LIN {X 0,Y 219.292,Z 411.491,A -85,B 0,C 180,E1 -21728.678,E2 -21728.678} C_VEL
LIN {X 0,Y 224.312,Z 397.889,A -85,B 0,C 180,E1 -21730.847,E2 -21730.847} C_VEL
LIN {X 0,Y 228.493,Z 384.244,A -85,B 0,C 180,E1 -21732.585,E2 -21732.585} C_VEL
LIN {X 0,Y 232.119,Z 370.098,A -85,B 0,C 180,E1 -21733.987,E2 -21733.987} C_VEL
LIN {X 0,Y 235.267,Z 355.521,A -85,B 0,C 180,E1 -21735.04,E2 -21735.04} C_VEL
LIN {X 0,Y 237.617,Z 340.528,A -85,B 0,C 180,E1 -21735.827,E2 -21735.827} C_VEL
LIN {X 0,Y 239.137,Z 325.025,A -85,B 0,C 180,E1 -21736.361,E2 -21736.361} C_VEL
LIN {X 0,Y 243.824,Z 251.846,A -85,B 0,C 180,E1 -21738.299,E2 -21738.299} C_VEL
LIN {X 0,Y 243.721,Z 250.513,A -85,B 0,C 180,E1 -21738.384,E2 -21738.384} C_VEL
LIN {X 0,Y 238.615,Z 238.715,A -85,B 0,C 180,E1 -21740.32,E2 -21740.32} C_VEL
LIN {X 0,Y 233.027,Z 227.32,A -85,B 0,C 180,E1 -21742.562,E2 -21742.562} C_VEL
LIN {X 0,Y 226.426,Z 215.296,A -85,B 0,C 180,E1 -21745.446,E2 -21745.446} C_VEL
LIN {X 0,Y 223.259,Z 210.38,A -85,B 0,C 180,E1 -21746.923,E2 -21746.923} C_VEL
LIN {X 0,Y 218.11,Z 203.18,A -85,B 0,C 180,E1 -21749.507,E2 -21749.507} C_VEL
LIN {X 0,Y 214.873,Z 198.917,A -85,B 0,C 180,E1 -21751.289,E2 -21751.289} C_VEL
LIN {X 0,Y 211.946,Z 195.104,A -85,B 0,C 180,E1 -21753.04,E2 -21753.04} C_VEL
LIN {X 0,Y 208.457,Z 191.041,A -85,B 0,C 180,E1 -21755.308,E2 -21755.308} C_VEL
LIN {X 0,Y 207.502,Z 189.433,A -85,B 0,C 180,E1 -21756.019,E2 -21756.019} C_VEL
LIN {X 0,Y 204.843,Z 187.038,A -85,B 0,C 180,E1 -21757.96,E2 -21757.96} C_VEL
LIN {X 0,Y 202.817,Z 183.879,A -85,B 0,C 180,E1 -21759.726,E2 -21759.726} C_VEL
LIN {X 0,Y 200.124,Z 181.801,A -85,B 0,C 180,E1 -21762.152,E2 -21762.152} C_VEL
LIN {X 0,Y 198.455,Z 178.926,A -85,B 0,C 180,E1 -21764.071,E2 -21764.071} C_VEL
LIN {X 0,Y 197.838,Z 178.138,A -85,B 0,C 180,E1 -21764.812,E2 -21764.812} C_VEL
LIN {X 0,Y 194.773,Z 176.058,A -85,B 0,C 180,E1 -21768.949,E2 -21768.949} C_VEL
LIN {X 0,Y 193.148,Z 172.89,A -85,B 0,C 180,E1 -21772.946,E2 -21772.946} C_VEL
LIN {X 0,Y 193.084,Z 172.118,A -85,B 0,C 180,E1 -21776.87,E2 -21776.87} C_VEL
LIN {X 0,Y 193.435,Z 172.028,A -85,B 0,C 180,E1 -21780,E2 -21780} C_VEL
LIN {X 0,Y 192.969,Z 172.206,A -85,B 0,C 180,E1 -21784.177,E2 -21784.177} C_VEL
LIN {X 0,Y 193.221,Z 173.073,A -85,B 0,C 180,E1 -21787.577,E2 -21787.577} C_VEL
LIN {X 0,Y 195.21,Z 176.548,A -85,B 0,C 180,E1 -21791.948,E2 -21791.948} C_VEL
LIN {X 0,Y 198.274,Z 178.589,A -85,B 0,C 180,E1 -21795.879,E2 -21795.879} C_VEL
LIN {X 0,Y 200,Z 181.766,A -85,B 0,C 180,E1 -21797.911,E2 -21797.911} C_VEL
LIN {X 0,Y 203.141,Z 184.315,A -85,B 0,C 180,E1 -21800.738,E2 -21800.738} C_VEL
LIN {X 0,Y 205.283,Z 187.689,A -85,B 0,C 180,E1 -21802.575,E2 -21802.575} C_VEL
LIN {X 0,Y 207.751,Z 189.895,A -85,B 0,C 180,E1 -21804.349,E2 -21804.349} C_VEL
LIN {X 0,Y 210.168,Z 193.303,A -85,B 0,C 180,E1 -21806.034,E2 -21806.034} C_VEL
LIN {X 0,Y 211.927,Z 195.13,A -85,B 0,C 180,E1 -21807.128,E2 -21807.128} C_VEL
LIN {X 0,Y 214.824,Z 198.894,A -85,B 0,C 180,E1 -21808.862,E2 -21808.862} C_VEL
LIN {X 0,Y 219.389,Z 204.99,A -85,B 0,C 180,E1 -21811.343,E2 -21811.343} C_VEL
LIN {X 0,Y 225.014,Z 212.914,A -85,B 0,C 180,E1 -21814.074,E2 -21814.074} C_VEL
LIN {X 0,Y 231.75,Z 223.28,A -85,B 0,C 180,E1 -21816.998,E2 -21816.998} C_VEL
LIN {X 0,Y 236.546,Z 232.253,A -85,B 0,C 180,E1 -21818.945,E2 -21818.945} C_VEL
LIN {X 0,Y 242.757,Z 245.504,A -85,B 0,C 180,E1 -21821.317,E2 -21821.317} C_VEL
LIN {X 0,Y 243.976,Z 248.447,A -85,B 0,C 180,E1 -21821.77,E2 -21821.77} C_VEL
LIN {X 0,Y 238.681,Z 329.958,A -85,B 0,C 180,E1 -21823.981,E2 -21823.981} C_VEL
LIN {X 0,Y 236.71,Z 345.1,A -85,B 0,C 180,E1 -21824.632,E2 -21824.632} C_VEL
LIN {X 0,Y 233.757,Z 361,A -85,B 0,C 180,E1 -21825.651,E2 -21825.651} C_VEL
LIN {X 0,Y 230.664,Z 374.454,A -85,B 0,C 180,E1 -21826.841,E2 -21826.841} C_VEL
LIN {X 0,Y 226.549,Z 389.137,A -85,B 0,C 180,E1 -21828.535,E2 -21828.535} C_VEL
LIN {X 0,Y 222.072,Z 402.265,A -85,B 0,C 180,E1 -21830.439,E2 -21830.439} C_VEL
LIN {X 0,Y 217.336,Z 414.499,A -85,B 0,C 180,E1 -21832.676,E2 -21832.676} C_VEL
LIN {X 0,Y 212.546,Z 425.648,A -85,B 0,C 180,E1 -21835.223,E2 -21835.223} C_VEL
LIN {X 0,Y 208.325,Z 435.023,A -85,B 0,C 180,E1 -21837.904,E2 -21837.904} C_VEL
LIN {X 0,Y 204.44,Z 443.018,A -85,B 0,C 180,E1 -21840.668,E2 -21840.668} C_VEL
LIN {X 0,Y 200.016,Z 451.913,A -85,B 0,C 180,E1 -21844.505,E2 -21844.505} C_VEL
LIN {X 0,Y 196.286,Z 459.241,A -85,B 0,C 180,E1 -21848.581,E2 -21848.581} C_VEL
LIN {X 0,Y 194.063,Z 464.117,A -85,B 0,C 180,E1 -21852.072,E2 -21852.072} C_VEL
LIN {X 0,Y 192.41,Z 467.578,A -85,B 0,C 180,E1 -21855.186,E2 -21855.186} C_VEL
LIN {X 0,Y 191.035,Z 471.08,A -85,B 0,C 180,E1 -21859.4,E2 -21859.4} C_VEL
LIN {X 0,Y 190.302,Z 473.393,A -85,B 0,C 180,E1 -21863.639,E2 -21863.639} C_VEL
LIN {X 0,Y 190.123,Z 474.569,A -85,B 0,C 180,E1 -21867.882,E2 -21867.882} C_VEL
LIN {X 0,Y 190.157,Z 474.726,A -85,B 0,C 180,E1 -21870,E2 -21870} C_VEL
LIN {X 0,Y 190.164,Z 474.157,A -85,B 0,C 180,E1 -21874.239,E2 -21874.239} C_VEL
LIN {X 0,Y 190.571,Z 472.465,A -85,B 0,C 180,E1 -21878.483,E2 -21878.483} C_VEL
LIN {X 0,Y 191.615,Z 469.61,A -85,B 0,C 180,E1 -21882.713,E2 -21882.713} C_VEL
LIN {X 0,Y 193.44,Z 465.523,A -85,B 0,C 180,E1 -21886.897,E2 -21886.897} C_VEL
LIN {X 0,Y 196.018,Z 460.105,A -85,B 0,C 180,E1 -21891.011,E2 -21891.011} C_VEL
LIN {X 0,Y 199.457,Z 453.203,A -85,B 0,C 180,E1 -21895.013,E2 -21895.013} C_VEL
LIN {X 0,Y 203.743,Z 444.589,A -85,B 0,C 180,E1 -21898.877,E2 -21898.877} C_VEL
LIN {X 0,Y 207.557,Z 436.846,A -85,B 0,C 180,E1 -21901.658,E2 -21901.658} C_VEL
LIN {X 0,Y 211.732,Z 427.731,A -85,B 0,C 180,E1 -21904.352,E2 -21904.352} C_VEL
LIN {X 0,Y 216.41,Z 416.978,A -85,B 0,C 180,E1 -21906.927,E2 -21906.927} C_VEL
LIN {X 0,Y 221.049,Z 405.24,A -85,B 0,C 180,E1 -21909.191,E2 -21909.191} C_VEL
LIN {X 0,Y 225.472,Z 392.675,A -85,B 0,C 180,E1 -21911.13,E2 -21911.13} C_VEL
LIN {X 0,Y 229.623,Z 378.937,A -85,B 0,C 180,E1 -21912.808,E2 -21912.808} C_VEL
LIN {X 0,Y 233.12,Z 364.473,A -85,B 0,C 180,E1 -21914.2,E2 -21914.2} C_VEL
LIN {X 0,Y 236.194,Z 349.03,A -85,B 0,C 180,E1 -21915.268,E2 -21915.268} C_VEL
LIN {X 0,Y 238.405,Z 333.558,A -85,B 0,C 180,E1 -21916.012,E2 -21916.012} C_VEL
LIN {X 0,Y 239.996,Z 314.021,A -85,B 0,C 180,E1 -21916.603,E2 -21916.603} C_VEL
LIN {X 0,Y 244.143,Z 248.635,A -85,B 0,C 180,E1 -21918.345,E2 -21918.345} C_VEL
LIN {X 0,Y 238.871,Z 236.861,A -85,B 0,C 180,E1 -21920.33,E2 -21920.33} C_VEL
LIN {X 0,Y 232.951,Z 225.151,A -85,B 0,C 180,E1 -21922.702,E2 -21922.702} C_VEL
LIN {X 0,Y 226.627,Z 215.259,A -85,B 0,C 180,E1 -21925.396,E2 -21925.396} C_VEL
LIN {X 0,Y 220.963,Z 207.127,A -85,B 0,C 180,E1 -21928.077,E2 -21928.077} C_VEL
LIN {X 0,Y 217.799,Z 202.785,A -85,B 0,C 180,E1 -21929.718,E2 -21929.718} C_VEL
LIN {X 0,Y 214.768,Z 198.812,A -85,B 0,C 180,E1 -21931.407,E2 -21931.407} C_VEL
LIN {X 0,Y 211.862,Z 194.934,A -85,B 0,C 180,E1 -21933.171,E2 -21933.171} C_VEL
LIN {X 0,Y 208.527,Z 191.176,A -85,B 0,C 180,E1 -21935.35,E2 -21935.35} C_VEL
LIN {X 0,Y 207.444,Z 189.425,A -85,B 0,C 180,E1 -21936.158,E2 -21936.158} C_VEL
LIN {X 0,Y 204.828,Z 187.087,A -85,B 0,C 180,E1 -21938.09,E2 -21938.09} C_VEL
LIN {X 0,Y 202.979,Z 183.958,A -85,B 0,C 180,E1 -21939.742,E2 -21939.742} C_VEL
LIN {X 0,Y 200.155,Z 181.908,A -85,B 0,C 180,E1 -21942.302,E2 -21942.302} C_VEL
LIN {X 0,Y 198.377,Z 178.846,A -85,B 0,C 180,E1 -21944.393,E2 -21944.393} C_VEL
LIN {X 0,Y 197.616,Z 178.027,A -85,B 0,C 180,E1 -21945.321,E2 -21945.321} C_VEL
LIN {X 0,Y 194.83,Z 176.101,A -85,B 0,C 180,E1 -21949.255,E2 -21949.255} C_VEL
LIN {X 0,Y 193.129,Z 172.939,A -85,B 0,C 180,E1 -21953.732,E2 -21953.732} C_VEL
LIN {X 0,Y 193.236,Z 172.108,A -85,B 0,C 180,E1 -21957.915,E2 -21957.915} C_VEL
LIN {X 0,Y 193.433,Z 172.045,A -85,B 0,C 180,E1 -21960,E2 -21960} C_VEL
LIN {X 0,Y 193.021,Z 172.37,A -85,B 0,C 180,E1 -21964.176,E2 -21964.176} C_VEL
LIN {X 0,Y 193.222,Z 173.274,A -85,B 0,C 180,E1 -21966.789,E2 -21966.789} C_VEL
LIN {X 0,Y 195.939,Z 177.12,A -85,B 0,C 180,E1 -21972.428,E2 -21972.428} C_VEL
LIN {X 0,Y 198.359,Z 178.653,A -85,B 0,C 180,E1 -21975.476,E2 -21975.476} C_VEL
LIN {X 0,Y 200.006,Z 181.652,A -85,B 0,C 180,E1 -21977.447,E2 -21977.447} C_VEL
LIN {X 0,Y 202.504,Z 183.704,A -85,B 0,C 180,E1 -21979.778,E2 -21979.778} C_VEL
LIN {X 0,Y 203.192,Z 184.29,A -85,B 0,C 180,E1 -21980.367,E2 -21980.367} C_VEL
LIN {X 0,Y 205.214,Z 187.529,A -85,B 0,C 180,E1 -21982.13,E2 -21982.13} C_VEL
LIN {X 0,Y 207.902,Z 189.993,A -85,B 0,C 180,E1 -21984.087,E2 -21984.087} C_VEL
LIN {X 0,Y 210.279,Z 193.339,A -85,B 0,C 180,E1 -21985.753,E2 -21985.753} C_VEL
LIN {X 0,Y 212.074,Z 195.266,A -85,B 0,C 180,E1 -21986.88,E2 -21986.88} C_VEL
LIN {X 0,Y 215.083,Z 199.099,A -85,B 0,C 180,E1 -21988.68,E2 -21988.68} C_VEL
LIN {X 0,Y 219.591,Z 205.175,A -85,B 0,C 180,E1 -21991.136,E2 -21991.136} C_VEL
LIN {X 0,Y 224.74,Z 212.412,A -85,B 0,C 180,E1 -21993.652,E2 -21993.652} C_VEL
LIN {X 0,Y 230.647,Z 222.756,A -85,B 0,C 180,E1 -21996.329,E2 -21996.329} C_VEL
LIN {X 0,Y 230.842,Z 223.057,A -85,B 0,C 180,E1 -21996.41,E2 -21996.41} C_VEL
LIN {X 0,Y 232.605,Z 227.635,A -85,B 0,C 180,E1 -21997.223,E2 -21997.223} C_VEL
LIN {X 0,Y 234.592,Z 236.333,A -85,B 0,C 180,E1 -21998.279,E2 -21998.279} C_VEL
LIN {X 0,Y 236.857,Z 247.053,A -85,B 0,C 180,E1 -21999.47,E2 -21999.47} C_VEL
LIN {X 0,Y 237.942,Z 250.365,A -85,B 0,C 180,E1 -21999.938,E2 -21999.938} C_VEL
LIN {X 0,Y 239.15,Z 253.343,A -85,B 0,C 180,E1 -22000.418,E2 -22000.418} C_VEL
LIN {X 0,Y 234.71,Z 321.37,A -85,B 0,C 180,E1 -22002.254,E2 -22002.254} C_VEL
LIN {X 0,Y 233.155,Z 338.204,A -85,B 0,C 180,E1 -22002.794,E2 -22002.794} C_VEL
LIN {X 0,Y 230.899,Z 353.15,A -85,B 0,C 180,E1 -22003.548,E2 -22003.548} C_VEL
LIN {X 0,Y 227.895,Z 367.197,A -85,B 0,C 180,E1 -22004.508,E2 -22004.508} C_VEL
LIN {X 0,Y 224.313,Z 381.084,A -85,B 0,C 180,E1 -22005.803,E2 -22005.803} C_VEL
LIN {X 0,Y 220.1,Z 394.817,A -85,B 0,C 180,E1 -22007.474,E2 -22007.474} C_VEL
LIN {X 0,Y 215.197,Z 408.195,A -85,B 0,C 180,E1 -22009.527,E2 -22009.527} C_VEL
LIN {X 0,Y 210.282,Z 419.992,A -85,B 0,C 180,E1 -22011.807,E2 -22011.807} C_VEL
LIN {X 0,Y 205.38,Z 430.801,A -85,B 0,C 180,E1 -22014.427,E2 -22014.427} C_VEL
LIN {X 0,Y 200.245,Z 441.405,A -85,B 0,C 180,E1 -22017.674,E2 -22017.674} C_VEL
LIN {X 0,Y 195.813,Z 450.086,A -85,B 0,C 180,E1 -22021.018,E2 -22021.018} C_VEL
LIN {X 0,Y 192.484,Z 456.43,A -85,B 0,C 180,E1 -22024.014,E2 -22024.014} C_VEL
LIN {X 0,Y 188.856,Z 463.389,A -85,B 0,C 180,E1 -22028.152,E2 -22028.152} C_VEL
LIN {X 0,Y 186.229,Z 468.861,A -85,B 0,C 180,E1 -22032.428,E2 -22032.428} C_VEL
LIN {X 0,Y 184.342,Z 472.997,A -85,B 0,C 180,E1 -22036.776,E2 -22036.776} C_VEL
LIN {X 0,Y 183.382,Z 475.897,A -85,B 0,C 180,E1 -22041.182,E2 -22041.182} C_VEL
LIN {X 0,Y 183.012,Z 477.625,A -85,B 0,C 180,E1 -22045.595,E2 -22045.595} C_VEL
LIN {X 0,Y 183.058,Z 478.215,A -85,B 0,C 180,E1 -22050,E2 -22050} C_VEL
LIN {X 0,Y 183.012,Z 477.609,A -85,B 0,C 180,E1 -22054.405,E2 -22054.405} C_VEL
LIN {X 0,Y 183.381,Z 475.859,A -85,B 0,C 180,E1 -22058.818,E2 -22058.818} C_VEL
LIN {X 0,Y 184.332,Z 472.943,A -85,B 0,C 180,E1 -22063.224,E2 -22063.224} C_VEL
LIN {X 0,Y 186.211,Z 468.793,A -85,B 0,C 180,E1 -22067.574,E2 -22067.574} C_VEL
LIN {X 0,Y 188.83,Z 463.295,A -85,B 0,C 180,E1 -22071.851,E2 -22071.851} C_VEL
LIN {X 0,Y 192.475,Z 456.304,A -85,B 0,C 180,E1 -22075.987,E2 -22075.987} C_VEL
LIN {X 0,Y 196.458,Z 448.827,A -85,B 0,C 180,E1 -22079.465,E2 -22079.465} C_VEL
LIN {X 0,Y 200.307,Z 440.84,A -85,B 0,C 180,E1 -22082.49,E2 -22082.49} C_VEL
LIN {X 0,Y 205.393,Z 430.604,A -85,B 0,C 180,E1 -22085.57,E2 -22085.57} C_VEL
LIN {X 0,Y 210.304,Z 419.758,A -85,B 0,C 180,E1 -22088.188,E2 -22088.188} C_VEL
LIN {X 0,Y 215.163,Z 407.916,A -85,B 0,C 180,E1 -22090.48,E2 -22090.48} C_VEL
LIN {X 0,Y 220.112,Z 394.443,A -85,B 0,C 180,E1 -22092.529,E2 -22092.529} C_VEL
LIN {X 0,Y 224.29,Z 380.638,A -85,B 0,C 180,E1 -22094.202,E2 -22094.202} C_VEL
LIN {X 0,Y 227.856,Z 366.64,A -85,B 0,C 180,E1 -22095.501,E2 -22095.501} C_VEL
LIN {X 0,Y 230.97,Z 351.645,A -85,B 0,C 180,E1 -22096.512,E2 -22096.512} C_VEL
LIN {X 0,Y 233.166,Z 337.075,A -85,B 0,C 180,E1 -22097.203,E2 -22097.203} C_VEL
LIN {X 0,Y 234.769,Z 317.786,A -85,B 0,C 180,E1 -22097.809,E2 -22097.809} C_VEL
LIN {X 0,Y 239.057,Z 253.811,A -85,B 0,C 180,E1 -22099.505,E2 -22099.505} C_VEL
LIN {X 0,Y 237.375,Z 249.287,A -85,B 0,C 180,E1 -22100.19,E2 -22100.19} C_VEL
LIN {X 0,Y 231.82,Z 236.957,A -85,B 0,C 180,E1 -22102.47,E2 -22102.47} C_VEL
LIN {X 0,Y 225.569,Z 224.712,A -85,B 0,C 180,E1 -22105.245,E2 -22105.245} C_VEL
LIN {X 0,Y 220.942,Z 216.873,A -85,B 0,C 180,E1 -22107.468,E2 -22107.468} C_VEL
LIN {X 0,Y 215.767,Z 209.397,A -85,B 0,C 180,E1 -22110.168,E2 -22110.168} C_VEL
LIN {X 0,Y 212.349,Z 204.879,A -85,B 0,C 180,E1 -22112.129,E2 -22112.129} C_VEL
LIN {X 0,Y 209.047,Z 200.53,A -85,B 0,C 180,E1 -22114.218,E2 -22114.218} C_VEL
LIN {X 0,Y 206.284,Z 197.099,A -85,B 0,C 180,E1 -22116.136,E2 -22116.136} C_VEL
LIN {X 0,Y 205.372,Z 195.826,A -85,B 0,C 180,E1 -22116.825,E2 -22116.825} C_VEL
LIN {X 0,Y 202.634,Z 192.917,A -85,B 0,C 180,E1 -22118.976,E2 -22118.976} C_VEL
LIN {X 0,Y 201.143,Z 190.555,A -85,B 0,C 180,E1 -22120.349,E2 -22120.349} C_VEL
LIN {X 0,Y 198.576,Z 188.38,A -85,B 0,C 180,E1 -22122.786,E2 -22122.786} C_VEL
LIN {X 0,Y 196.671,Z 185.074,A -85,B 0,C 180,E1 -22125.117,E2 -22125.117} C_VEL
LIN {X 0,Y 193.651,Z 182.936,A -85,B 0,C 180,E1 -22129.347,E2 -22129.347} C_VEL
LIN {X 0,Y 191.942,Z 179.766,A -85,B 0,C 180,E1 -22133.43,E2 -22133.43} C_VEL
LIN {X 0,Y 190.91,Z 178.77,A -85,B 0,C 180,E1 -22137.891,E2 -22137.891} C_VEL
LIN {X 0,Y 190.889,Z 178.767,A -85,B 0,C 180,E1 -22142.11,E2 -22142.11} C_VEL
LIN {X 0,Y 192.003,Z 179.832,A -85,B 0,C 180,E1 -22146.921,E2 -22146.921} C_VEL
LIN {X 0,Y 194.313,Z 183.638,A -85,B 0,C 180,E1 -22151.937,E2 -22151.937} C_VEL
LIN {X 0,Y 196.86,Z 185.396,A -85,B 0,C 180,E1 -22155.307,E2 -22155.307} C_VEL
LIN {X 0,Y 198.783,Z 188.745,A -85,B 0,C 180,E1 -22157.624,E2 -22157.624} C_VEL
LIN {X 0,Y 201.508,Z 191.037,A -85,B 0,C 180,E1 -22160.164,E2 -22160.164} C_VEL
LIN {X 0,Y 203.775,Z 194.502,A -85,B 0,C 180,E1 -22162.162,E2 -22162.162} C_VEL
LIN {X 0,Y 205.859,Z 196.44,A -85,B 0,C 180,E1 -22163.717,E2 -22163.717} C_VEL
LIN {X 0,Y 208.564,Z 200.115,A -85,B 0,C 180,E1 -22165.65,E2 -22165.65} C_VEL
LIN {X 0,Y 209.923,Z 201.694,A -85,B 0,C 180,E1 -22166.535,E2 -22166.535} C_VEL
LIN {X 0,Y 213.72,Z 206.734,A -85,B 0,C 180,E1 -22168.86,E2 -22168.86} C_VEL
LIN {X 0,Y 217.46,Z 211.932,A -85,B 0,C 180,E1 -22170.935,E2 -22170.935} C_VEL
LIN {X 0,Y 222.021,Z 218.436,A -85,B 0,C 180,E1 -22173.232,E2 -22173.232} C_VEL
LIN {X 0,Y 228.588,Z 228.837,A -85,B 0,C 180,E1 -22176.22,E2 -22176.22} C_VEL
LIN {X 0,Y 232.998,Z 237.37,A -85,B 0,C 180,E1 -22178.1,E2 -22178.1} C_VEL
LIN {X 0,Y 238.901,Z 250.316,A -85,B 0,C 180,E1 -22180.469,E2 -22180.469} C_VEL
LIN {X 0,Y 239.153,Z 251.863,A -85,B 0,C 180,E1 -22180.61,E2 -22180.61} C_VEL
LIN {X 0,Y 233.807,Z 330.039,A -85,B 0,C 180,E1 -22182.729,E2 -22182.729} C_VEL
LIN {X 0,Y 231.659,Z 345.951,A -85,B 0,C 180,E1 -22183.431,E2 -22183.431} C_VEL
LIN {X 0,Y 228.733,Z 361.074,A -85,B 0,C 180,E1 -22184.408,E2 -22184.408} C_VEL
LIN {X 0,Y 225.536,Z 374.526,A -85,B 0,C 180,E1 -22185.607,E2 -22185.607} C_VEL
LIN {X 0,Y 221.613,Z 388.162,A -85,B 0,C 180,E1 -22187.18,E2 -22187.18} C_VEL
LIN {X 0,Y 217.098,Z 401.091,A -85,B 0,C 180,E1 -22189.039,E2 -22189.039} C_VEL
LIN {X 0,Y 212.119,Z 413.53,A -85,B 0,C 180,E1 -22191.29,E2 -22191.29} C_VEL
LIN {X 0,Y 207.508,Z 423.947,A -85,B 0,C 180,E1 -22193.651,E2 -22193.651} C_VEL
LIN {X 0,Y 202.936,Z 433.612,A -85,B 0,C 180,E1 -22196.351,E2 -22196.351} C_VEL
LIN {X 0,Y 198.947,Z 441.859,A -85,B 0,C 180,E1 -22199.188,E2 -22199.188} C_VEL
LIN {X 0,Y 194.682,Z 449.971,A -85,B 0,C 180,E1 -22202.595,E2 -22202.595} C_VEL
LIN {X 0,Y 191.095,Z 456.666,A -85,B 0,C 180,E1 -22206.137,E2 -22206.137} C_VEL
LIN {X 0,Y 187.879,Z 462.862,A -85,B 0,C 180,E1 -22210.326,E2 -22210.326} C_VEL
LIN {X 0,Y 185.512,Z 467.646,A -85,B 0,C 180,E1 -22214.622,E2 -22214.622} C_VEL
LIN {X 0,Y 184.04,Z 471.147,A -85,B 0,C 180,E1 -22218.993,E2 -22218.993} C_VEL
LIN {X 0,Y 183.232,Z 473.46,A -85,B 0,C 180,E1 -22223.393,E2 -22223.393} C_VEL
LIN {X 0,Y 183.041,Z 474.636,A -85,B 0,C 180,E1 -22227.8,E2 -22227.8} C_VEL
LIN {X 0,Y 183.068,Z 474.792,A -85,B 0,C 180,E1 -22230,E2 -22230} C_VEL
LIN {X 0,Y 183.078,Z 474.223,A -85,B 0,C 180,E1 -22234.403,E2 -22234.403} C_VEL
LIN {X 0,Y 183.534,Z 472.531,A -85,B 0,C 180,E1 -22238.811,E2 -22238.811} C_VEL
LIN {X 0,Y 184.668,Z 469.676,A -85,B 0,C 180,E1 -22243.2,E2 -22243.2} C_VEL
LIN {X 0,Y 186.615,Z 465.588,A -85,B 0,C 180,E1 -22247.535,E2 -22247.535} C_VEL
LIN {X 0,Y 189.53,Z 459.81,A -85,B 0,C 180,E1 -22252.023,E2 -22252.023} C_VEL
LIN {X 0,Y 192.992,Z 453.268,A -85,B 0,C 180,E1 -22255.912,E2 -22255.912} C_VEL
LIN {X 0,Y 197.525,Z 444.654,A -85,B 0,C 180,E1 -22259.876,E2 -22259.876} C_VEL
LIN {X 0,Y 200.862,Z 438.293,A -85,B 0,C 180,E1 -22262.234,E2 -22262.234} C_VEL
LIN {X 0,Y 205.126,Z 429.42,A -85,B 0,C 180,E1 -22265.021,E2 -22265.021} C_VEL
LIN {X 0,Y 209.92,Z 418.99,A -85,B 0,C 180,E1 -22267.662,E2 -22267.662} C_VEL
LIN {X 0,Y 214.708,Z 407.645,A -85,B 0,C 180,E1 -22269.97,E2 -22269.97} C_VEL
LIN {X 0,Y 219.302,Z 395.318,A -85,B 0,C 180,E1 -22271.989,E2 -22271.989} C_VEL
LIN {X 0,Y 223.648,Z 381.836,A -85,B 0,C 180,E1 -22273.736,E2 -22273.736} C_VEL
LIN {X 0,Y 227.334,Z 367.862,A -85,B 0,C 180,E1 -22275.163,E2 -22275.163} C_VEL
LIN {X 0,Y 230.476,Z 353.504,A -85,B 0,C 180,E1 -22276.246,E2 -22276.246} C_VEL
LIN {X 0,Y 233.017,Z 338.009,A -85,B 0,C 180,E1 -22277.084,E2 -22277.084} C_VEL
LIN {X 0,Y 234.572,Z 322.858,A -85,B 0,C 180,E1 -22277.623,E2 -22277.623} C_VEL
LIN {X 0,Y 239.359,Z 251.323,A -85,B 0,C 180,E1 -22279.529,E2 -22279.529} C_VEL
LIN {X 0,Y 234.599,Z 240.563,A -85,B 0,C 180,E1 -22281.428,E2 -22281.428} C_VEL
LIN {X 0,Y 229.419,Z 230.11,A -85,B 0,C 180,E1 -22283.621,E2 -22283.621} C_VEL
LIN {X 0,Y 223.515,Z 220.68,A -85,B 0,C 180,E1 -22286.263,E2 -22286.263} C_VEL
LIN {X 0,Y 218.485,Z 213.239,A -85,B 0,C 180,E1 -22288.755,E2 -22288.755} C_VEL
LIN {X 0,Y 215.01,Z 208.427,A -85,B 0,C 180,E1 -22290.639,E2 -22290.639} C_VEL
LIN {X 0,Y 212.443,Z 204.96,A -85,B 0,C 180,E1 -22292.142,E2 -22292.142} C_VEL
LIN {X 0,Y 209.155,Z 200.66,A -85,B 0,C 180,E1 -22294.232,E2 -22294.232} C_VEL
LIN {X 0,Y 206.371,Z 197.247,A -85,B 0,C 180,E1 -22296.173,E2 -22296.173} C_VEL
LIN {X 0,Y 205.346,Z 195.837,A -85,B 0,C 180,E1 -22296.954,E2 -22296.954} C_VEL
LIN {X 0,Y 202.705,Z 193.053,A -85,B 0,C 180,E1 -22299.05,E2 -22299.05} C_VEL
LIN {X 0,Y 201.308,Z 190.663,A -85,B 0,C 180,E1 -22300.365,E2 -22300.365} C_VEL
LIN {X 0,Y 198.655,Z 188.536,A -85,B 0,C 180,E1 -22302.897,E2 -22302.897} C_VEL
LIN {X 0,Y 196.771,Z 185.147,A -85,B 0,C 180,E1 -22305.257,E2 -22305.257} C_VEL
LIN {X 0,Y 193.774,Z 183.052,A -85,B 0,C 180,E1 -22309.552,E2 -22309.552} C_VEL
LIN {X 0,Y 191.949,Z 179.786,A -85,B 0,C 180,E1 -22314.221,E2 -22314.221} C_VEL
LIN {X 0,Y 191.221,Z 178.897,A -85,B 0,C 180,E1 -22317.893,E2 -22317.893} C_VEL
LIN {X 0,Y 191.232,Z 178.897,A -85,B 0,C 180,E1 -22322.106,E2 -22322.106} C_VEL
LIN {X 0,Y 192.125,Z 180.108,A -85,B 0,C 180,E1 -22326.3,E2 -22326.3} C_VEL
LIN {X 0,Y 194.911,Z 184.113,A -85,B 0,C 180,E1 -22332.23,E2 -22332.23} C_VEL
LIN {X 0,Y 196.933,Z 185.341,A -85,B 0,C 180,E1 -22334.862,E2 -22334.862} C_VEL
LIN {X 0,Y 198.609,Z 188.405,A -85,B 0,C 180,E1 -22336.957,E2 -22336.957} C_VEL
LIN {X 0,Y 201.013,Z 190.483,A -85,B 0,C 180,E1 -22339.293,E2 -22339.293} C_VEL
LIN {X 0,Y 201.736,Z 191.396,A -85,B 0,C 180,E1 -22339.962,E2 -22339.962} C_VEL
LIN {X 0,Y 204.215,Z 194.854,A -85,B 0,C 180,E1 -22342.111,E2 -22342.111} C_VEL
LIN {X 0,Y 206.063,Z 196.647,A -85,B 0,C 180,E1 -22343.494,E2 -22343.494} C_VEL
LIN {X 0,Y 208.755,Z 200.236,A -85,B 0,C 180,E1 -22345.419,E2 -22345.419} C_VEL
LIN {X 0,Y 210.208,Z 201.994,A -85,B 0,C 180,E1 -22346.372,E2 -22346.372} C_VEL
LIN {X 0,Y 213.833,Z 206.786,A -85,B 0,C 180,E1 -22348.595,E2 -22348.595} C_VEL
LIN {X 0,Y 217.456,Z 211.781,A -85,B 0,C 180,E1 -22350.615,E2 -22350.615} C_VEL
LIN {X 0,Y 222.087,Z 218.452,A -85,B 0,C 180,E1 -22352.965,E2 -22352.965} C_VEL
LIN {X 0,Y 227.929,Z 229.093,A -85,B 0,C 180,E1 -22355.727,E2 -22355.727} C_VEL
LIN {X 0,Y 233.778,Z 240.945,A -85,B 0,C 180,E1 -22358.25,E2 -22358.25} C_VEL
LIN {X 0,Y 237.942,Z 250.365,A -85,B 0,C 180,E1 -22359.938,E2 -22359.938} C_VEL
LIN {X 0,Y 238.326,Z 252.647,A -85,B 0,C 180,E1 -22360.153,E2 -22360.153} C_VEL
LIN {X 0,Y 237.865,Z 256.466,A -85,B 0,C 180,E1 -22360.196,E2 -22360.196} C_VEL
LIN {X 0,Y 236.707,Z 260.242,A -85,B 0,C 180,E1 -22360.039,E2 -22360.039} C_VEL
LIN {X 0,Y 234.28,Z 266.935,A -85,B 0,C 180,E1 -22359.644,E2 -22359.644} C_VEL
LIN {X 0,Y 233.477,Z 271.147,A -85,B 0,C 180,E1 -22359.605,E2 -22359.605} C_VEL
LIN {X 0,Y 229.082,Z 332.406,A -85,B 0,C 180,E1 -22361.268,E2 -22361.268} C_VEL
LIN {X 0,Y 227.071,Z 347.712,A -85,B 0,C 180,E1 -22361.945,E2 -22361.945} C_VEL
LIN {X 0,Y 224.09,Z 362.557,A -85,B 0,C 180,E1 -22362.853,E2 -22362.853} C_VEL
LIN {X 0,Y 220.265,Z 377.464,A -85,B 0,C 180,E1 -22364.118,E2 -22364.118} C_VEL
LIN {X 0,Y 216.069,Z 391.39,A -85,B 0,C 180,E1 -22365.728,E2 -22365.728} C_VEL
LIN {X 0,Y 211.311,Z 404.581,A -85,B 0,C 180,E1 -22367.662,E2 -22367.662} C_VEL
LIN {X 0,Y 206.068,Z 416.966,A -85,B 0,C 180,E1 -22369.929,E2 -22369.929} C_VEL
LIN {X 0,Y 200.437,Z 429.107,A -85,B 0,C 180,E1 -22372.782,E2 -22372.782} C_VEL
LIN {X 0,Y 195.341,Z 439.324,A -85,B 0,C 180,E1 -22375.842,E2 -22375.842} C_VEL
LIN {X 0,Y 190.275,Z 448.902,A -85,B 0,C 180,E1 -22379.478,E2 -22379.478} C_VEL
LIN {X 0,Y 186.052,Z 456.364,A -85,B 0,C 180,E1 -22383.045,E2 -22383.045} C_VEL
LIN {X 0,Y 182.219,Z 463.323,A -85,B 0,C 180,E1 -22387.313,E2 -22387.313} C_VEL
LIN {X 0,Y 179.398,Z 468.795,A -85,B 0,C 180,E1 -22391.735,E2 -22391.735} C_VEL
LIN {X 0,Y 177.383,Z 472.931,A -85,B 0,C 180,E1 -22396.248,E2 -22396.248} C_VEL
LIN {X 0,Y 176.327,Z 475.831,A -85,B 0,C 180,E1 -22400.826,E2 -22400.826} C_VEL
LIN {X 0,Y 175.933,Z 477.559,A -85,B 0,C 180,E1 -22405.417,E2 -22405.417} C_VEL
LIN {X 0,Y 175.971,Z 478.149,A -85,B 0,C 180,E1 -22410,E2 -22410} C_VEL
LIN {X 0,Y 175.933,Z 477.542,A -85,B 0,C 180,E1 -22414.582,E2 -22414.582} C_VEL
LIN {X 0,Y 176.326,Z 475.792,A -85,B 0,C 180,E1 -22419.174,E2 -22419.174} C_VEL
LIN {X 0,Y 177.372,Z 472.875,A -85,B 0,C 180,E1 -22423.753,E2 -22423.753} C_VEL
LIN {X 0,Y 179.378,Z 468.725,A -85,B 0,C 180,E1 -22428.267,E2 -22428.267} C_VEL
LIN {X 0,Y 182.197,Z 463.227,A -85,B 0,C 180,E1 -22432.689,E2 -22432.689} C_VEL
LIN {X 0,Y 186.043,Z 456.235,A -85,B 0,C 180,E1 -22436.957,E2 -22436.957} C_VEL
LIN {X 0,Y 190.267,Z 448.758,A -85,B 0,C 180,E1 -22440.523,E2 -22440.523} C_VEL
LIN {X 0,Y 194.632,Z 440.142,A -85,B 0,C 180,E1 -22443.849,E2 -22443.849} C_VEL
LIN {X 0,Y 199.616,Z 430.534,A -85,B 0,C 180,E1 -22446.765,E2 -22446.765} C_VEL
LIN {X 0,Y 204.736,Z 419.688,A -85,B 0,C 180,E1 -22449.424,E2 -22449.424} C_VEL
LIN {X 0,Y 209.801,Z 407.846,A -85,B 0,C 180,E1 -22451.742,E2 -22451.742} C_VEL
LIN {X 0,Y 214.787,Z 394.746,A -85,B 0,C 180,E1 -22453.76,E2 -22453.76} C_VEL
LIN {X 0,Y 219.24,Z 380.566,A -85,B 0,C 180,E1 -22455.5,E2 -22455.5} C_VEL
LIN {X 0,Y 222.93,Z 366.567,A -85,B 0,C 180,E1 -22456.805,E2 -22456.805} C_VEL
LIN {X 0,Y 226.152,Z 351.569,A -85,B 0,C 180,E1 -22457.815,E2 -22457.815} C_VEL
LIN {X 0,Y 228.412,Z 336.995,A -85,B 0,C 180,E1 -22458.507,E2 -22458.507} C_VEL
LIN {X 0,Y 230.061,Z 317.698,A -85,B 0,C 180,E1 -22459.119,E2 -22459.119} C_VEL
LIN {X 0,Y 234.327,Z 255.848,A -85,B 0,C 180,E1 -22460.778,E2 -22460.778} C_VEL
LIN {X 0,Y 229.106,Z 243.706,A -85,B 0,C 180,E1 -22463.015,E2 -22463.015} C_VEL
LIN {X 0,Y 224.33,Z 233.88,A -85,B 0,C 180,E1 -22465.196,E2 -22465.196} C_VEL
LIN {X 0,Y 218.838,Z 223.545,A -85,B 0,C 180,E1 -22467.934,E2 -22467.934} C_VEL
LIN {X 0,Y 213.028,Z 215.078,A -85,B 0,C 180,E1 -22471.084,E2 -22471.084} C_VEL
LIN {X 0,Y 210.145,Z 211.143,A -85,B 0,C 180,E1 -22472.822,E2 -22472.822} C_VEL
LIN {X 0,Y 206.848,Z 206.734,A -85,B 0,C 180,E1 -22475.002,E2 -22475.002} C_VEL
LIN {X 0,Y 204.119,Z 203.095,A -85,B 0,C 180,E1 -22477.01,E2 -22477.01} C_VEL
LIN {X 0,Y 200.559,Z 198.847,A -85,B 0,C 180,E1 -22479.955,E2 -22479.955} C_VEL
LIN {X 0,Y 199.494,Z 197.222,A -85,B 0,C 180,E1 -22480.982,E2 -22480.982} C_VEL
LIN {X 0,Y 197.06,Z 194.953,A -85,B 0,C 180,E1 -22483.423,E2 -22483.423} C_VEL
LIN {X 0,Y 195.308,Z 191.864,A -85,B 0,C 180,E1 -22485.677,E2 -22485.677} C_VEL
LIN {X 0,Y 192.551,Z 189.83,A -85,B 0,C 180,E1 -22489.729,E2 -22489.729} C_VEL
LIN {X 0,Y 190.989,Z 186.757,A -85,B 0,C 180,E1 -22493.662,E2 -22493.662} C_VEL
LIN {X 0,Y 190.045,Z 185.824,A -85,B 0,C 180,E1 -22497.881,E2 -22497.881} C_VEL
LIN {X 0,Y 190.024,Z 185.82,A -85,B 0,C 180,E1 -22502.12,E2 -22502.12} C_VEL
LIN {X 0,Y 191.087,Z 186.893,A -85,B 0,C 180,E1 -22506.812,E2 -22506.812} C_VEL
LIN {X 0,Y 193.173,Z 190.535,A -85,B 0,C 180,E1 -22511.543,E2 -22511.543} C_VEL
LIN {X 0,Y 195.511,Z 192.177,A -85,B 0,C 180,E1 -22514.774,E2 -22514.774} C_VEL
LIN {X 0,Y 197.344,Z 195.443,A -85,B 0,C 180,E1 -22517.086,E2 -22517.086} C_VEL
LIN {X 0,Y 199.932,Z 197.827,A -85,B 0,C 180,E1 -22519.618,E2 -22519.618} C_VEL
LIN {X 0,Y 202.268,Z 201.272,A -85,B 0,C 180,E1 -22521.732,E2 -22521.732} C_VEL
LIN {X 0,Y 204.138,Z 203.208,A -85,B 0,C 180,E1 -22523.189,E2 -22523.189} C_VEL
LIN {X 0,Y 207.03,Z 206.974,A -85,B 0,C 180,E1 -22525.301,E2 -22525.301} C_VEL
LIN {X 0,Y 211.383,Z 212.854,A -85,B 0,C 180,E1 -22528.12,E2 -22528.12} C_VEL
LIN {X 0,Y 216.684,Z 220.381,A -85,B 0,C 180,E1 -22531.126,E2 -22531.126} C_VEL
LIN {X 0,Y 223.433,Z 230.929,A -85,B 0,C 180,E1 -22534.485,E2 -22534.485} C_VEL
LIN {X 0,Y 227.567,Z 238.371,A -85,B 0,C 180,E1 -22536.367,E2 -22536.367} C_VEL
LIN {X 0,Y 233.709,Z 251.733,A -85,B 0,C 180,E1 -22539.016,E2 -22539.016} C_VEL
LIN {X 0,Y 234.438,Z 253.545,A -85,B 0,C 180,E1 -22539.322,E2 -22539.322} C_VEL
LIN {X 0,Y 229.053,Z 330.121,A -85,B 0,C 180,E1 -22541.426,E2 -22541.426} C_VEL
LIN {X 0,Y 226.844,Z 346.027,A -85,B 0,C 180,E1 -22542.13,E2 -22542.13} C_VEL
LIN {X 0,Y 223.836,Z 361.147,A -85,B 0,C 180,E1 -22543.113,E2 -22543.113} C_VEL
LIN {X 0,Y 220.207,Z 375.681,A -85,B 0,C 180,E1 -22544.43,E2 -22544.43} C_VEL
LIN {X 0,Y 215.942,Z 389.759,A -85,B 0,C 180,E1 -22546.107,E2 -22546.107} C_VEL
LIN {X 0,Y 211.297,Z 402.406,A -85,B 0,C 180,E1 -22547.981,E2 -22547.981} C_VEL
LIN {X 0,Y 206.16,Z 414.639,A -85,B 0,C 180,E1 -22550.269,E2 -22550.269} C_VEL
LIN {X 0,Y 200.992,Z 425.787,A -85,B 0,C 180,E1 -22552.902,E2 -22552.902} C_VEL
LIN {X 0,Y 195.612,Z 436.646,A -85,B 0,C 180,E1 -22556.175,E2 -22556.175} C_VEL
LIN {X 0,Y 190.772,Z 445.604,A -85,B 0,C 180,E1 -22559.566,E2 -22559.566} C_VEL
LIN {X 0,Y 186.655,Z 453.054,A -85,B 0,C 180,E1 -22563.139,E2 -22563.139} C_VEL
LIN {X 0,Y 182.649,Z 460.114,A -85,B 0,C 180,E1 -22567.441,E2 -22567.441} C_VEL
LIN {X 0,Y 179.857,Z 465.489,A -85,B 0,C 180,E1 -22571.784,E2 -22571.784} C_VEL
LIN {X 0,Y 177.746,Z 469.617,A -85,B 0,C 180,E1 -22576.276,E2 -22576.276} C_VEL
LIN {X 0,Y 176.538,Z 472.515,A -85,B 0,C 180,E1 -22580.837,E2 -22580.837} C_VEL
LIN {X 0,Y 176.009,Z 474.254,A -85,B 0,C 180,E1 -22585.42,E2 -22585.42} C_VEL
LIN {X 0,Y 175.981,Z 474.859,A -85,B 0,C 180,E1 -22590,E2 -22590} C_VEL
LIN {X 0,Y 176.008,Z 474.29,A -85,B 0,C 180,E1 -22594.581,E2 -22594.581} C_VEL
LIN {X 0,Y 176.49,Z 472.597,A -85,B 0,C 180,E1 -22599.165,E2 -22599.165} C_VEL
LIN {X 0,Y 177.72,Z 469.742,A -85,B 0,C 180,E1 -22603.726,E2 -22603.726} C_VEL
LIN {X 0,Y 179.819,Z 465.654,A -85,B 0,C 180,E1 -22608.22,E2 -22608.22} C_VEL
LIN {X 0,Y 182.729,Z 460.236,A -85,B 0,C 180,E1 -22612.62,E2 -22612.62} C_VEL
LIN {X 0,Y 186.585,Z 453.334,A -85,B 0,C 180,E1 -22616.872,E2 -22616.872} C_VEL
LIN {X 0,Y 191.384,Z 444.718,A -85,B 0,C 180,E1 -22620.938,E2 -22620.938} C_VEL
LIN {X 0,Y 195.343,Z 437.298,A -85,B 0,C 180,E1 -22623.746,E2 -22623.746} C_VEL
LIN {X 0,Y 200.11,Z 427.859,A -85,B 0,C 180,E1 -22626.659,E2 -22626.659} C_VEL
LIN {X 0,Y 205.17,Z 417.105,A -85,B 0,C 180,E1 -22629.325,E2 -22629.325} C_VEL
LIN {X 0,Y 210.189,Z 405.365,A -85,B 0,C 180,E1 -22631.648,E2 -22631.648} C_VEL
LIN {X 0,Y 215.279,Z 391.95,A -85,B 0,C 180,E1 -22633.737,E2 -22633.737} C_VEL
LIN {X 0,Y 219.585,Z 378.388,A -85,B 0,C 180,E1 -22635.409,E2 -22635.409} C_VEL
LIN {X 0,Y 223.155,Z 364.591,A -85,B 0,C 180,E1 -22636.744,E2 -22636.744} C_VEL
LIN {X 0,Y 226.444,Z 349.142,A -85,B 0,C 180,E1 -22637.816,E2 -22637.816} C_VEL
LIN {X 0,Y 228.783,Z 333.661,A -85,B 0,C 180,E1 -22638.568,E2 -22638.568} C_VEL
LIN {X 0,Y 230.497,Z 314.107,A -85,B 0,C 180,E1 -22639.161,E2 -22639.161} C_VEL
LIN {X 0,Y 234.589,Z 253.767,A -85,B 0,C 180,E1 -22640.8,E2 -22640.8} C_VEL
LIN {X 0,Y 229.418,Z 242.043,A -85,B 0,C 180,E1 -22643.008,E2 -22643.008} C_VEL
LIN {X 0,Y 225.15,Z 233.647,A -85,B 0,C 180,E1 -22644.932,E2 -22644.932} C_VEL
LIN {X 0,Y 218.598,Z 223.137,A -85,B 0,C 180,E1 -22648.098,E2 -22648.098} C_VEL
LIN {X 0,Y 213.023,Z 215.017,A -85,B 0,C 180,E1 -22651.151,E2 -22651.151} C_VEL
LIN {X 0,Y 210.195,Z 211.167,A -85,B 0,C 180,E1 -22652.867,E2 -22652.867} C_VEL
LIN {X 0,Y 206.962,Z 206.871,A -85,B 0,C 180,E1 -22655.017,E2 -22655.017} C_VEL
LIN {X 0,Y 204.175,Z 203.163,A -85,B 0,C 180,E1 -22657.082,E2 -22657.082} C_VEL
LIN {X 0,Y 200.638,Z 199.031,A -85,B 0,C 180,E1 -22660.03,E2 -22660.03} C_VEL
LIN {X 0,Y 199.66,Z 197.373,A -85,B 0,C 180,E1 -22660.998,E2 -22660.998} C_VEL
LIN {X 0,Y 197.104,Z 195.063,A -85,B 0,C 180,E1 -22663.585,E2 -22663.585} C_VEL
LIN {X 0,Y 195.312,Z 191.916,A -85,B 0,C 180,E1 -22665.943,E2 -22665.943} C_VEL
LIN {X 0,Y 192.612,Z 189.852,A -85,B 0,C 180,E1 -22670.071,E2 -22670.071} C_VEL
LIN {X 0,Y 191.009,Z 186.779,A -85,B 0,C 180,E1 -22674.457,E2 -22674.457} C_VEL
LIN {X 0,Y 190.356,Z 185.953,A -85,B 0,C 180,E1 -22677.884,E2 -22677.884} C_VEL
LIN {X 0,Y 190.429,Z 186.042,A -85,B 0,C 180,E1 -22682.644,E2 -22682.644} C_VEL
LIN {X 0,Y 191.175,Z 187.11,A -85,B 0,C 180,E1 -22686.067,E2 -22686.067} C_VEL
LIN {X 0,Y 193.721,Z 190.974,A -85,B 0,C 180,E1 -22691.775,E2 -22691.775} C_VEL
LIN {X 0,Y 195.612,Z 192.249,A -85,B 0,C 180,E1 -22694.367,E2 -22694.367} C_VEL
LIN {X 0,Y 197.644,Z 195.663,A -85,B 0,C 180,E1 -22696.926,E2 -22696.926} C_VEL
LIN {X 0,Y 199.931,Z 197.692,A -85,B 0,C 180,E1 -22699.175,E2 -22699.175} C_VEL
LIN {X 0,Y 202.487,Z 201.409,A -85,B 0,C 180,E1 -22701.506,E2 -22701.506} C_VEL
LIN {X 0,Y 204.222,Z 203.192,A -85,B 0,C 180,E1 -22702.865,E2 -22702.865} C_VEL
LIN {X 0,Y 207.24,Z 207.113,A -85,B 0,C 180,E1 -22705.081,E2 -22705.081} C_VEL
LIN {X 0,Y 211.772,Z 213.311,A -85,B 0,C 180,E1 -22708.021,E2 -22708.021} C_VEL
LIN {X 0,Y 215.187,Z 218.152,A -85,B 0,C 180,E1 -22709.999,E2 -22709.999} C_VEL
LIN {X 0,Y 219.817,Z 225.219,A -85,B 0,C 180,E1 -22712.448,E2 -22712.448} C_VEL
LIN {X 0,Y 225.074,Z 235.191,A -85,B 0,C 180,E1 -22715.038,E2 -22715.038} C_VEL
LIN {X 0,Y 230.288,Z 246.097,A -85,B 0,C 180,E1 -22717.397,E2 -22717.397} C_VEL
LIN {X 0,Y 234.413,Z 255.832,A -85,B 0,C 180,E1 -22719.159,E2 -22719.159} C_VEL
LIN {X 0,Y 233.477,Z 271.147,A -85,B 0,C 180,E1 -22719.605,E2 -22719.605} C_VEL
LIN {X 0,Y 232.645,Z 276.996,A -85,B 0,C 180,E1 -22719.635,E2 -22719.635} C_VEL
LIN {X 0,Y 227.648,Z 296.051,A -85,B 0,C 180,E1 -22719.037,E2 -22719.037} C_VEL
LIN {X 0,Y 226.804,Z 301.902,A -85,B 0,C 180,E1 -22719.063,E2 -22719.063} C_VEL
LIN {X 0,Y 224.316,Z 333.54,A -85,B 0,C 180,E1 -22719.948,E2 -22719.948} C_VEL
LIN {X 0,Y 222.095,Z 349.226,A -85,B 0,C 180,E1 -22720.67,E2 -22720.67} C_VEL
LIN {X 0,Y 219.046,Z 363.688,A -85,B 0,C 180,E1 -22721.585,E2 -22721.585} C_VEL
LIN {X 0,Y 215.375,Z 377.403,A -85,B 0,C 180,E1 -22722.759,E2 -22722.759} C_VEL
LIN {X 0,Y 211.024,Z 391.329,A -85,B 0,C 180,E1 -22724.378,E2 -22724.378} C_VEL
LIN {X 0,Y 206.103,Z 404.518,A -85,B 0,C 180,E1 -22726.329,E2 -22726.329} C_VEL
LIN {X 0,Y 200.672,Z 416.903,A -85,B 0,C 180,E1 -22728.62,E2 -22728.62} C_VEL
LIN {X 0,Y 194.798,Z 429.043,A -85,B 0,C 180,E1 -22731.512,E2 -22731.512} C_VEL
LIN {X 0,Y 189.85,Z 438.441,A -85,B 0,C 180,E1 -22734.348,E2 -22734.348} C_VEL
LIN {X 0,Y 184.829,Z 447.627,A -85,B 0,C 180,E1 -22737.836,E2 -22737.836} C_VEL
LIN {X 0,Y 180.298,Z 455.289,A -85,B 0,C 180,E1 -22741.477,E2 -22741.477} C_VEL
LIN {X 0,Y 176.559,Z 461.642,A -85,B 0,C 180,E1 -22745.294,E2 -22745.294} C_VEL
LIN {X 0,Y 173.288,Z 467.483,A -85,B 0,C 180,E1 -22749.834,E2 -22749.834} C_VEL
LIN {X 0,Y 171.45,Z 470.957,A -85,B 0,C 180,E1 -22753.325,E2 -22753.325} C_VEL
LIN {X 0,Y 169.765,Z 474.465,A -85,B 0,C 180,E1 -22758.054,E2 -22758.054} C_VEL
LIN {X 0,Y 168.964,Z 476.771,A -85,B 0,C 180,E1 -22762.832,E2 -22762.832} C_VEL
LIN {X 0,Y 168.787,Z 477.93,A -85,B 0,C 180,E1 -22767.614,E2 -22767.614} C_VEL
LIN {X 0,Y 168.868,Z 478.082,A -85,B 0,C 180,E1 -22770,E2 -22770} C_VEL
LIN {X 0,Y 168.85,Z 477.476,A -85,B 0,C 180,E1 -22774.775,E2 -22774.775} C_VEL
LIN {X 0,Y 169.292,Z 475.725,A -85,B 0,C 180,E1 -22779.559,E2 -22779.559} C_VEL
LIN {X 0,Y 170.431,Z 472.808,A -85,B 0,C 180,E1 -22784.325,E2 -22784.325} C_VEL
LIN {X 0,Y 172.578,Z 468.657,A -85,B 0,C 180,E1 -22789.013,E2 -22789.013} C_VEL
LIN {X 0,Y 175.597,Z 463.158,A -85,B 0,C 180,E1 -22793.593,E2 -22793.593} C_VEL
LIN {X 0,Y 179.699,Z 456.167,A -85,B 0,C 180,E1 -22797.99,E2 -22797.99} C_VEL
LIN {X 0,Y 184.145,Z 448.69,A -85,B 0,C 180,E1 -22801.653,E2 -22801.653} C_VEL
LIN {X 0,Y 188.994,Z 439.637,A -85,B 0,C 180,E1 -22805.212,E2 -22805.212} C_VEL
LIN {X 0,Y 194.81,Z 428.83,A -85,B 0,C 180,E1 -22808.485,E2 -22808.485} C_VEL
LIN {X 0,Y 200.637,Z 416.634,A -85,B 0,C 180,E1 -22811.388,E2 -22811.388} C_VEL
LIN {X 0,Y 206.106,Z 404.197,A -85,B 0,C 180,E1 -22813.67,E2 -22813.67} C_VEL
LIN {X 0,Y 210.942,Z 391.126,A -85,B 0,C 180,E1 -22815.601,E2 -22815.601} C_VEL
LIN {X 0,Y 215.386,Z 376.886,A -85,B 0,C 180,E1 -22817.237,E2 -22817.237} C_VEL
LIN {X 0,Y 219.001,Z 363.099,A -85,B 0,C 180,E1 -22818.428,E2 -22818.428} C_VEL
LIN {X 0,Y 222.171,Z 347.633,A -85,B 0,C 180,E1 -22819.394,E2 -22819.394} C_VEL
LIN {X 0,Y 224.289,Z 332.598,A -85,B 0,C 180,E1 -22820.04,E2 -22820.04} C_VEL
LIN {X 0,Y 229.739,Z 259.058,A -85,B 0,C 180,E1 -22822.037,E2 -22822.037} C_VEL
LIN {X 0,Y 229.194,Z 257.047,A -85,B 0,C 180,E1 -22822.312,E2 -22822.312} C_VEL
LIN {X 0,Y 223.495,Z 243.949,A -85,B 0,C 180,E1 -22824.95,E2 -22824.95} C_VEL
LIN {X 0,Y 217.299,Z 231.607,A -85,B 0,C 180,E1 -22828.089,E2 -22828.089} C_VEL
LIN {X 0,Y 213.544,Z 225.398,A -85,B 0,C 180,E1 -22830.147,E2 -22830.147} C_VEL
LIN {X 0,Y 208.314,Z 217.75,A -85,B 0,C 180,E1 -22833.316,E2 -22833.316} C_VEL
LIN {X 0,Y 204.848,Z 213.124,A -85,B 0,C 180,E1 -22835.688,E2 -22835.688} C_VEL
LIN {X 0,Y 201.701,Z 208.839,A -85,B 0,C 180,E1 -22838.137,E2 -22838.137} C_VEL
LIN {X 0,Y 198.969,Z 205.513,A -85,B 0,C 180,E1 -22840.528,E2 -22840.528} C_VEL
LIN {X 0,Y 198.131,Z 204.052,A -85,B 0,C 180,E1 -22841.383,E2 -22841.383} C_VEL
LIN {X 0,Y 195.65,Z 201.658,A -85,B 0,C 180,E1 -22843.97,E2 -22843.97} C_VEL
LIN {X 0,Y 194.054,Z 198.775,A -85,B 0,C 180,E1 -22846.117,E2 -22846.117} C_VEL
LIN {X 0,Y 191.406,Z 196.645,A -85,B 0,C 180,E1 -22850.223,E2 -22850.223} C_VEL
LIN {X 0,Y 189.961,Z 193.63,A -85,B 0,C 180,E1 -22854.161,E2 -22854.161} C_VEL
LIN {X 0,Y 189.059,Z 192.704,A -85,B 0,C 180,E1 -22860,E2 -22860} C_VEL
LIN {X 0,Y 189.988,Z 193.664,A -85,B 0,C 180,E1 -22866.105,E2 -22866.105} C_VEL
LIN {X 0,Y 192.158,Z 197.534,A -85,B 0,C 180,E1 -22871.338,E2 -22871.338} C_VEL
LIN {X 0,Y 194.199,Z 199.065,A -85,B 0,C 180,E1 -22874.273,E2 -22874.273} C_VEL
LIN {X 0,Y 196.146,Z 202.39,A -85,B 0,C 180,E1 -22876.791,E2 -22876.791} C_VEL
LIN {X 0,Y 198.349,Z 204.531,A -85,B 0,C 180,E1 -22879.032,E2 -22879.032} C_VEL
LIN {X 0,Y 200.915,Z 208.186,A -85,B 0,C 180,E1 -22881.414,E2 -22881.414} C_VEL
LIN {X 0,Y 202.368,Z 209.829,A -85,B 0,C 180,E1 -22882.594,E2 -22882.594} C_VEL
LIN {X 0,Y 206.05,Z 214.81,A -85,B 0,C 180,E1 -22885.35,E2 -22885.35} C_VEL
LIN {X 0,Y 209.466,Z 219.549,A -85,B 0,C 180,E1 -22887.609,E2 -22887.609} C_VEL
LIN {X 0,Y 214.332,Z 226.72,A -85,B 0,C 180,E1 -22890.479,E2 -22890.479} C_VEL
LIN {X 0,Y 220.311,Z 236.292,A -85,B 0,C 180,E1 -22893.592,E2 -22893.592} C_VEL
LIN {X 0,Y 224.083,Z 243.202,A -85,B 0,C 180,E1 -22895.399,E2 -22895.399} C_VEL
LIN {X 0,Y 229.869,Z 256.241,A -85,B 0,C 180,E1 -22898.04,E2 -22898.04} C_VEL
LIN {X 0,Y 224.493,Z 329.639,A -85,B 0,C 180,E1 -22900.05,E2 -22900.05} C_VEL
LIN {X 0,Y 222.294,Z 345.33,A -85,B 0,C 180,E1 -22900.73,E2 -22900.73} C_VEL
LIN {X 0,Y 219.061,Z 361.221,A -85,B 0,C 180,E1 -22901.762,E2 -22901.762} C_VEL
LIN {X 0,Y 215.822,Z 373.887,A -85,B 0,C 180,E1 -22902.888,E2 -22902.888} C_VEL
LIN {X 0,Y 211.828,Z 387.004,A -85,B 0,C 180,E1 -22904.397,E2 -22904.397} C_VEL
LIN {X 0,Y 207.077,Z 399.942,A -85,B 0,C 180,E1 -22906.25,E2 -22906.25} C_VEL
LIN {X 0,Y 201.663,Z 412.603,A -85,B 0,C 180,E1 -22908.536,E2 -22908.536} C_VEL
LIN {X 0,Y 196.211,Z 424.086,A -85,B 0,C 180,E1 -22911.184,E2 -22911.184} C_VEL
LIN {X 0,Y 191.215,Z 433.75,A -85,B 0,C 180,E1 -22913.98,E2 -22913.98} C_VEL
LIN {X 0,Y 186.11,Z 443.224,A -85,B 0,C 180,E1 -22917.445,E2 -22917.445} C_VEL
LIN {X 0,Y 181.502,Z 451.113,A -85,B 0,C 180,E1 -22921.052,E2 -22921.052} C_VEL
LIN {X 0,Y 177.08,Z 458.479,A -85,B 0,C 180,E1 -22925.372,E2 -22925.372} C_VEL
LIN {X 0,Y 173.763,Z 464.32,A -85,B 0,C 180,E1 -22929.892,E2 -22929.892} C_VEL
LIN {X 0,Y 171.79,Z 467.781,A -85,B 0,C 180,E1 -22933.359,E2 -22933.359} C_VEL
LIN {X 0,Y 170.05,Z 471.282,A -85,B 0,C 180,E1 -22938.074,E2 -22938.074} C_VEL
LIN {X 0,Y 169.11,Z 473.593,A -85,B 0,C 180,E1 -22942.838,E2 -22942.838} C_VEL
LIN {X 0,Y 168.859,Z 474.769,A -85,B 0,C 180,E1 -22947.615,E2 -22947.615} C_VEL
LIN {X 0,Y 168.88,Z 474.925,A -85,B 0,C 180,E1 -22950,E2 -22950} C_VEL
LIN {X 0,Y 168.931,Z 474.356,A -85,B 0,C 180,E1 -22954.773,E2 -22954.773} C_VEL
LIN {X 0,Y 169.467,Z 472.663,A -85,B 0,C 180,E1 -22959.549,E2 -22959.549} C_VEL
LIN {X 0,Y 170.776,Z 469.808,A -85,B 0,C 180,E1 -22964.295,E2 -22964.295} C_VEL
LIN {X 0,Y 173.049,Z 465.72,A -85,B 0,C 180,E1 -22968.96,E2 -22968.96} C_VEL
LIN {X 0,Y 176.148,Z 460.302,A -85,B 0,C 180,E1 -22973.515,E2 -22973.515} C_VEL
LIN {X 0,Y 180.237,Z 453.399,A -85,B 0,C 180,E1 -22977.899,E2 -22977.899} C_VEL
LIN {X 0,Y 185.321,Z 444.783,A -85,B 0,C 180,E1 -22982.068,E2 -22982.068} C_VEL
LIN {X 0,Y 189.291,Z 437.629,A -85,B 0,C 180,E1 -22984.85,E2 -22984.85} C_VEL
LIN {X 0,Y 194.427,Z 427.923,A -85,B 0,C 180,E1 -22987.916,E2 -22987.916} C_VEL
LIN {X 0,Y 199.709,Z 417.168,A -85,B 0,C 180,E1 -22990.62,E2 -22990.62} C_VEL
LIN {X 0,Y 204.932,Z 405.428,A -85,B 0,C 180,E1 -22992.969,E2 -22992.969} C_VEL
LIN {X 0,Y 210.137,Z 392.204,A -85,B 0,C 180,E1 -22995.048,E2 -22995.048} C_VEL
LIN {X 0,Y 214.66,Z 378.449,A -85,B 0,C 180,E1 -22996.758,E2 -22996.758} C_VEL
LIN {X 0,Y 218.356,Z 364.65,A -85,B 0,C 180,E1 -22998.099,E2 -22998.099} C_VEL
LIN {X 0,Y 221.749,Z 349.198,A -85,B 0,C 180,E1 -22999.173,E2 -22999.173} C_VEL
LIN {X 0,Y 224.159,Z 333.712,A -85,B 0,C 180,E1 -22999.925,E2 -22999.925} C_VEL
LIN {X 0,Y 225.929,Z 314.149,A -85,B 0,C 180,E1 -23000.52,E2 -23000.52} C_VEL
LIN {X 0,Y 229.99,Z 256.353,A -85,B 0,C 180,E1 -23002.1,E2 -23002.1} C_VEL
LIN {X 0,Y 224.321,Z 243.54,A -85,B 0,C 180,E1 -23004.694,E2 -23004.694} C_VEL
LIN {X 0,Y 220.733,Z 236.886,A -85,B 0,C 180,E1 -23006.415,E2 -23006.415} C_VEL
LIN {X 0,Y 215.005,Z 227.682,A -85,B 0,C 180,E1 -23009.38,E2 -23009.38} C_VEL
LIN {X 0,Y 210.244,Z 220.539,A -85,B 0,C 180,E1 -23012.161,E2 -23012.161} C_VEL
LIN {X 0,Y 207.815,Z 217.182,A -85,B 0,C 180,E1 -23013.715,E2 -23013.715} C_VEL
LIN {X 0,Y 204.853,Z 213.092,A -85,B 0,C 180,E1 -23015.79,E2 -23015.79} C_VEL
LIN {X 0,Y 201.799,Z 208.985,A -85,B 0,C 180,E1 -23018.184,E2 -23018.184} C_VEL
LIN {X 0,Y 198.996,Z 205.581,A -85,B 0,C 180,E1 -23020.664,E2 -23020.664} C_VEL
LIN {X 0,Y 197.916,Z 203.944,A -85,B 0,C 180,E1 -23021.764,E2 -23021.764} C_VEL
LIN {X 0,Y 195.425,Z 201.333,A -85,B 0,C 180,E1 -23024.484,E2 -23024.484} C_VEL
LIN {X 0,Y 194.071,Z 198.815,A -85,B 0,C 180,E1 -23026.385,E2 -23026.385} C_VEL
LIN {X 0,Y 191.514,Z 196.722,A -85,B 0,C 180,E1 -23030.495,E2 -23030.495} C_VEL
LIN {X 0,Y 190.072,Z 193.773,A -85,B 0,C 180,E1 -23034.696,E2 -23034.696} C_VEL
LIN {X 0,Y 189.49,Z 193.005,A -85,B 0,C 180,E1 -23037.874,E2 -23037.874} C_VEL
LIN {X 0,Y 189.501,Z 193,A -85,B 0,C 180,E1 -23042.125,E2 -23042.125} C_VEL
LIN {X 0,Y 190.231,Z 194.085,A -85,B 0,C 180,E1 -23045.831,E2 -23045.831} C_VEL
LIN {X 0,Y 192.701,Z 197.968,A -85,B 0,C 180,E1 -23051.571,E2 -23051.571} C_VEL
LIN {X 0,Y 194.31,Z 199.124,A -85,B 0,C 180,E1 -23053.864,E2 -23053.864} C_VEL
LIN {X 0,Y 196.446,Z 202.608,A -85,B 0,C 180,E1 -23056.631,E2 -23056.631} C_VEL
LIN {X 0,Y 198.454,Z 204.569,A -85,B 0,C 180,E1 -23058.686,E2 -23058.686} C_VEL
LIN {X 0,Y 201.206,Z 208.405,A -85,B 0,C 180,E1 -23061.247,E2 -23061.247} C_VEL
LIN {X 0,Y 202.511,Z 209.847,A -85,B 0,C 180,E1 -23062.307,E2 -23062.307} C_VEL
LIN {X 0,Y 206.269,Z 215.009,A -85,B 0,C 180,E1 -23065.14,E2 -23065.14} C_VEL
LIN {X 0,Y 209.819,Z 219.929,A -85,B 0,C 180,E1 -23067.488,E2 -23067.488} C_VEL
LIN {X 0,Y 214.096,Z 226.169,A -85,B 0,C 180,E1 -23070.02,E2 -23070.02} C_VEL
LIN {X 0,Y 217.484,Z 231.756,A -85,B 0,C 180,E1 -23071.872,E2 -23071.872} C_VEL
LIN {X 0,Y 223.15,Z 243.134,A -85,B 0,C 180,E1 -23074.77,E2 -23074.77} C_VEL
LIN {X 0,Y 228.417,Z 254.911,A -85,B 0,C 180,E1 -23077.23,E2 -23077.23} C_VEL
LIN {X 0,Y 229.901,Z 258.651,A -85,B 0,C 180,E1 -23077.899,E2 -23077.899} C_VEL
LIN {X 0,Y 226.804,Z 301.902,A -85,B 0,C 180,E1 -23079.063,E2 -23079.063} C_VEL
LIN {X 0,Y 225.976,Z 307.754,A -85,B 0,C 180,E1 -23079.085,E2 -23079.085} C_VEL
LIN {X 0,Y 220.953,Z 326.794,A -85,B 0,C 180,E1 -23078.453,E2 -23078.453} C_VEL
LIN {X 0,Y 219.953,Z 332.616,A -85,B 0,C 180,E1 -23078.504,E2 -23078.504} C_VEL
LIN {X 0,Y 217.694,Z 348.407,A -85,B 0,C 180,E1 -23079.212,E2 -23079.212} C_VEL
LIN {X 0,Y 214.686,Z 362.44,A -85,B 0,C 180,E1 -23080.074,E2 -23080.074} C_VEL
LIN {X 0,Y 210.621,Z 377.343,A -85,B 0,C 180,E1 -23081.342,E2 -23081.342} C_VEL
LIN {X 0,Y 206.31,Z 390.631,A -85,B 0,C 180,E1 -23082.878,E2 -23082.878} C_VEL
LIN {X 0,Y 201.011,Z 404.456,A -85,B 0,C 180,E1 -23084.927,E2 -23084.927} C_VEL
LIN {X 0,Y 195.383,Z 416.84,A -85,B 0,C 180,E1 -23087.239,E2 -23087.239} C_VEL
LIN {X 0,Y 189.261,Z 428.978,A -85,B 0,C 180,E1 -23090.166,E2 -23090.166} C_VEL
LIN {X 0,Y 183.434,Z 439.549,A -85,B 0,C 180,E1 -23093.454,E2 -23093.454} C_VEL
LIN {X 0,Y 178.099,Z 448.772,A -85,B 0,C 180,E1 -23097.14,E2 -23097.14} C_VEL
LIN {X 0,Y 173.433,Z 456.234,A -85,B 0,C 180,E1 -23100.904,E2 -23100.904} C_VEL
LIN {X 0,Y 169.108,Z 463.192,A -85,B 0,C 180,E1 -23105.443,E2 -23105.443} C_VEL
LIN {X 0,Y 165.841,Z 468.663,A -85,B 0,C 180,E1 -23110.182,E2 -23110.182} C_VEL
LIN {X 0,Y 163.519,Z 472.798,A -85,B 0,C 180,E1 -23115.056,E2 -23115.056} C_VEL
LIN {X 0,Y 162.246,Z 475.698,A -85,B 0,C 180,E1 -23120.022,E2 -23120.022} C_VEL
LIN {X 0,Y 161.749,Z 477.426,A -85,B 0,C 180,E1 -23125.015,E2 -23125.015} C_VEL
LIN {X 0,Y 161.772,Z 478.016,A -85,B 0,C 180,E1 -23130,E2 -23130} C_VEL
LIN {X 0,Y 161.749,Z 477.409,A -85,B 0,C 180,E1 -23134.985,E2 -23134.985} C_VEL
LIN {X 0,Y 162.244,Z 475.658,A -85,B 0,C 180,E1 -23139.978,E2 -23139.978} C_VEL
LIN {X 0,Y 163.507,Z 472.74,A -85,B 0,C 180,E1 -23144.945,E2 -23144.945} C_VEL
LIN {X 0,Y 165.821,Z 468.589,A -85,B 0,C 180,E1 -23149.82,E2 -23149.82} C_VEL
LIN {X 0,Y 169.05,Z 463.09,A -85,B 0,C 180,E1 -23154.566,E2 -23154.566} C_VEL
LIN {X 0,Y 173.426,Z 456.098,A -85,B 0,C 180,E1 -23159.097,E2 -23159.097} C_VEL
LIN {X 0,Y 178.092,Z 448.621,A -85,B 0,C 180,E1 -23162.862,E2 -23162.862} C_VEL
LIN {X 0,Y 183.019,Z 439.87,A -85,B 0,C 180,E1 -23166.391,E2 -23166.391} C_VEL
LIN {X 0,Y 188.366,Z 430.396,A -85,B 0,C 180,E1 -23169.366,E2 -23169.366} C_VEL
LIN {X 0,Y 193.9,Z 419.548,A -85,B 0,C 180,E1 -23172.109,E2 -23172.109} C_VEL
LIN {X 0,Y 199.403,Z 407.706,A -85,B 0,C 180,E1 -23174.467,E2 -23174.467} C_VEL
LIN {X 0,Y 204.682,Z 394.75,A -85,B 0,C 180,E1 -23176.498,E2 -23176.498} C_VEL
LIN {X 0,Y 209.506,Z 380.422,A -85,B 0,C 180,E1 -23178.279,E2 -23178.279} C_VEL
LIN {X 0,Y 213.462,Z 366.42,A -85,B 0,C 180,E1 -23179.585,E2 -23179.585} C_VEL
LIN {X 0,Y 216.85,Z 351.418,A -85,B 0,C 180,E1 -23180.603,E2 -23180.603} C_VEL
LIN {X 0,Y 219.302,Z 336.573,A -85,B 0,C 180,E1 -23181.295,E2 -23181.295} C_VEL
LIN {X 0,Y 221.088,Z 316.93,A -85,B 0,C 180,E1 -23181.914,E2 -23181.914} C_VEL
LIN {X 0,Y 225.225,Z 261.023,A -85,B 0,C 180,E1 -23183.427,E2 -23183.427} C_VEL
LIN {X 0,Y 220.078,Z 248.814,A -85,B 0,C 180,E1 -23185.956,E2 -23185.956} C_VEL
LIN {X 0,Y 214.228,Z 236.761,A -85,B 0,C 180,E1 -23189.099,E2 -23189.099} C_VEL
LIN {X 0,Y 210.464,Z 230.524,A -85,B 0,C 180,E1 -23191.279,E2 -23191.279} C_VEL
LIN {X 0,Y 206.078,Z 223.925,A -85,B 0,C 180,E1 -23194.091,E2 -23194.091} C_VEL
LIN {X 0,Y 202.88,Z 219.494,A -85,B 0,C 180,E1 -23196.388,E2 -23196.388} C_VEL
LIN {X 0,Y 199.836,Z 215.256,A -85,B 0,C 180,E1 -23198.871,E2 -23198.871} C_VEL
LIN {X 0,Y 197.164,Z 211.755,A -85,B 0,C 180,E1 -23201.356,E2 -23201.356} C_VEL
LIN {X 0,Y 196.275,Z 210.519,A -85,B 0,C 180,E1 -23202.281,E2 -23202.281} C_VEL
LIN {X 0,Y 193.866,Z 207.761,A -85,B 0,C 180,E1 -23205.031,E2 -23205.031} C_VEL
LIN {X 0,Y 192.817,Z 205.641,A -85,B 0,C 180,E1 -23206.564,E2 -23206.564} C_VEL
LIN {X 0,Y 190.41,Z 203.637,A -85,B 0,C 180,E1 -23210.439,E2 -23210.439} C_VEL
LIN {X 0,Y 189.018,Z 200.624,A -85,B 0,C 180,E1 -23214.399,E2 -23214.399} C_VEL
LIN {X 0,Y 188.194,Z 199.753,A -85,B 0,C 180,E1 -23220,E2 -23220} C_VEL
LIN {X 0,Y 189.044,Z 200.657,A -85,B 0,C 180,E1 -23225.868,E2 -23225.868} C_VEL
LIN {X 0,Y 190.997,Z 204.383,A -85,B 0,C 180,E1 -23230.87,E2 -23230.87} C_VEL
LIN {X 0,Y 192.917,Z 205.953,A -85,B 0,C 180,E1 -23233.783,E2 -23233.783} C_VEL
LIN {X 0,Y 194.95,Z 209.36,A -85,B 0,C 180,E1 -23236.493,E2 -23236.493} C_VEL
LIN {X 0,Y 196.828,Z 211.273,A -85,B 0,C 180,E1 -23238.475,E2 -23238.475} C_VEL
LIN {X 0,Y 199.481,Z 215.022,A -85,B 0,C 180,E1 -23241.018,E2 -23241.018} C_VEL
LIN {X 0,Y 200.762,Z 216.645,A -85,B 0,C 180,E1 -23242.106,E2 -23242.106} C_VEL
LIN {X 0,Y 204.127,Z 221.296,A -85,B 0,C 180,E1 -23244.723,E2 -23244.723} C_VEL
LIN {X 0,Y 207.278,Z 225.815,A -85,B 0,C 180,E1 -23246.9,E2 -23246.9} C_VEL
LIN {X 0,Y 211.922,Z 232.863,A -85,B 0,C 180,E1 -23249.763,E2 -23249.763} C_VEL
LIN {X 0,Y 217.416,Z 241.953,A -85,B 0,C 180,E1 -23252.762,E2 -23252.762} C_VEL
LIN {X 0,Y 220.897,Z 248.632,A -85,B 0,C 180,E1 -23254.522,E2 -23254.522} C_VEL
LIN {X 0,Y 225.348,Z 258.948,A -85,B 0,C 180,E1 -23256.683,E2 -23256.683} C_VEL
LIN {X 0,Y 219.9,Z 330.563,A -85,B 0,C 180,E1 -23258.668,E2 -23258.668} C_VEL
LIN {X 0,Y 217.594,Z 346.18,A -85,B 0,C 180,E1 -23259.362,E2 -23259.362} C_VEL
LIN {X 0,Y 214.389,Z 361.295,A -85,B 0,C 180,E1 -23260.344,E2 -23260.344} C_VEL
LIN {X 0,Y 210.506,Z 375.825,A -85,B 0,C 180,E1 -23261.667,E2 -23261.667} C_VEL
LIN {X 0,Y 206.128,Z 389.386,A -85,B 0,C 180,E1 -23263.292,E2 -23263.292} C_VEL
LIN {X 0,Y 200.972,Z 402.546,A -85,B 0,C 180,E1 -23265.27,E2 -23265.27} C_VEL
LIN {X 0,Y 195.408,Z 414.779,A -85,B 0,C 180,E1 -23267.596,E2 -23267.596} C_VEL
LIN {X 0,Y 189.802,Z 425.926,A -85,B 0,C 180,E1 -23270.303,E2 -23270.303} C_VEL
LIN {X 0,Y 184.496,Z 435.607,A -85,B 0,C 180,E1 -23273.274,E2 -23273.274} C_VEL
LIN {X 0,Y 180.154,Z 443.293,A -85,B 0,C 180,E1 -23276.227,E2 -23276.227} C_VEL
LIN {X 0,Y 175.272,Z 451.182,A -85,B 0,C 180,E1 -23279.919,E2 -23279.919} C_VEL
LIN {X 0,Y 170.612,Z 458.547,A -85,B 0,C 180,E1 -23284.372,E2 -23284.372} C_VEL
LIN {X 0,Y 167.043,Z 464.389,A -85,B 0,C 180,E1 -23289.046,E2 -23289.046} C_VEL
LIN {X 0,Y 164.974,Z 467.848,A -85,B 0,C 180,E1 -23292.65,E2 -23292.65} C_VEL
LIN {X 0,Y 163.087,Z 471.349,A -85,B 0,C 180,E1 -23297.557,E2 -23297.557} C_VEL
LIN {X 0,Y 162.042,Z 473.66,A -85,B 0,C 180,E1 -23302.524,E2 -23302.524} C_VEL
LIN {X 0,Y 161.762,Z 474.855,A -85,B 0,C 180,E1 -23307.818,E2 -23307.818} C_VEL
LIN {X 0,Y 161.765,Z 474.864,A -85,B 0,C 180,E1 -23312.21,E2 -23312.21} C_VEL
LIN {X 0,Y 162.032,Z 473.718,A -85,B 0,C 180,E1 -23317.477,E2 -23317.477} C_VEL
LIN {X 0,Y 163.07,Z 471.45,A -85,B 0,C 180,E1 -23322.444,E2 -23322.444} C_VEL
LIN {X 0,Y 164.948,Z 467.989,A -85,B 0,C 180,E1 -23327.353,E2 -23327.353} C_VEL
LIN {X 0,Y 167.828,Z 463.251,A -85,B 0,C 180,E1 -23332.141,E2 -23332.141} C_VEL
LIN {X 0,Y 171.658,Z 457.114,A -85,B 0,C 180,E1 -23336.767,E2 -23336.767} C_VEL
LIN {X 0,Y 176.47,Z 449.387,A -85,B 0,C 180,E1 -23341.18,E2 -23341.18} C_VEL
LIN {X 0,Y 181.593,Z 441.15,A -85,B 0,C 180,E1 -23344.81,E2 -23344.81} C_VEL
LIN {X 0,Y 186.261,Z 432.725,A -85,B 0,C 180,E1 -23347.817,E2 -23347.817} C_VEL
LIN {X 0,Y 191.561,Z 422.841,A -85,B 0,C 180,E1 -23350.633,E2 -23350.633} C_VEL
LIN {X 0,Y 196.779,Z 412.155,A -85,B 0,C 180,E1 -23353.083,E2 -23353.083} C_VEL
LIN {X 0,Y 202.372,Z 399.385,A -85,B 0,C 180,E1 -23355.392,E2 -23355.392} C_VEL
LIN {X 0,Y 207.226,Z 386.543,A -85,B 0,C 180,E1 -23357.224,E2 -23357.224} C_VEL
LIN {X 0,Y 211.465,Z 373.008,A -85,B 0,C 180,E1 -23358.759,E2 -23358.759} C_VEL
LIN {X 0,Y 214.865,Z 360.165,A -85,B 0,C 180,E1 -23359.869,E2 -23359.869} C_VEL
LIN {X 0,Y 218.074,Z 344.623,A -85,B 0,C 180,E1 -23360.844,E2 -23360.844} C_VEL
LIN {X 0,Y 220.195,Z 329.679,A -85,B 0,C 180,E1 -23361.491,E2 -23361.491} C_VEL
LIN {X 0,Y 225.494,Z 258.98,A -85,B 0,C 180,E1 -23363.457,E2 -23363.457} C_VEL
LIN {X 0,Y 220.298,Z 247.171,A -85,B 0,C 180,E1 -23365.994,E2 -23365.994} C_VEL
LIN {X 0,Y 216.176,Z 239.703,A -85,B 0,C 180,E1 -23368.109,E2 -23368.109} C_VEL
LIN {X 0,Y 211.054,Z 231.364,A -85,B 0,C 180,E1 -23370.992,E2 -23370.992} C_VEL
LIN {X 0,Y 206.192,Z 224.015,A -85,B 0,C 180,E1 -23374.106,E2 -23374.106} C_VEL
LIN {X 0,Y 202.854,Z 219.45,A -85,B 0,C 180,E1 -23376.52,E2 -23376.52} C_VEL
LIN {X 0,Y 199.972,Z 215.468,A -85,B 0,C 180,E1 -23378.891,E2 -23378.891} C_VEL
LIN {X 0,Y 197.119,Z 211.671,A -85,B 0,C 180,E1 -23381.586,E2 -23381.586} C_VEL
LIN {X 0,Y 196.451,Z 210.7,A -85,B 0,C 180,E1 -23382.297,E2 -23382.297} C_VEL
LIN {X 0,Y 193.998,Z 207.941,A -85,B 0,C 180,E1 -23385.121,E2 -23385.121} C_VEL
LIN {X 0,Y 192.841,Z 205.714,A -85,B 0,C 180,E1 -23386.833,E2 -23386.833} C_VEL
LIN {X 0,Y 190.352,Z 203.466,A -85,B 0,C 180,E1 -23391.097,E2 -23391.097} C_VEL
LIN {X 0,Y 189.075,Z 200.669,A -85,B 0,C 180,E1 -23395.202,E2 -23395.202} C_VEL
LIN {X 0,Y 188.522,Z 199.872,A -85,B 0,C 180,E1 -23400,E2 -23400} C_VEL
LIN {X 0,Y 189.095,Z 200.693,A -85,B 0,C 180,E1 -23404.797,E2 -23404.797} C_VEL
LIN {X 0,Y 191.846,Z 205.084,A -85,B 0,C 180,E1 -23411.624,E2 -23411.624} C_VEL
LIN {X 0,Y 193.067,Z 206.055,A -85,B 0,C 180,E1 -23413.418,E2 -23413.418} C_VEL
LIN {X 0,Y 195.331,Z 209.64,A -85,B 0,C 180,E1 -23416.42,E2 -23416.42} C_VEL
LIN {X 0,Y 196.933,Z 211.276,A -85,B 0,C 180,E1 -23418.118,E2 -23418.118} C_VEL
LIN {X 0,Y 199.72,Z 215.175,A -85,B 0,C 180,E1 -23420.805,E2 -23420.805} C_VEL
LIN {X 0,Y 200.837,Z 216.576,A -85,B 0,C 180,E1 -23421.759,E2 -23421.759} C_VEL
LIN {X 0,Y 204.068,Z 221.056,A -85,B 0,C 180,E1 -23424.303,E2 -23424.303} C_VEL
LIN {X 0,Y 207.595,Z 226.159,A -85,B 0,C 180,E1 -23426.758,E2 -23426.758} C_VEL
LIN {X 0,Y 211.633,Z 232.213,A -85,B 0,C 180,E1 -23429.261,E2 -23429.261} C_VEL
LIN {X 0,Y 214.63,Z 237.398,A -85,B 0,C 180,E1 -23430.987,E2 -23430.987} C_VEL
LIN {X 0,Y 219.692,Z 247.809,A -85,B 0,C 180,E1 -23433.721,E2 -23433.721} C_VEL
LIN {X 0,Y 224.761,Z 259.567,A -85,B 0,C 180,E1 -23436.235,E2 -23436.235} C_VEL
LIN {X 0,Y 225.416,Z 261.223,A -85,B 0,C 180,E1 -23436.547,E2 -23436.547} C_VEL
LIN {X 0,Y 219.953,Z 332.616,A -85,B 0,C 180,E1 -23438.504,E2 -23438.504} C_VEL
LIN {X 0,Y 218.823,Z 338.417,A -85,B 0,C 180,E1 -23438.583,E2 -23438.583} C_VEL
LIN {X 0,Y 215.558,Z 347.778,A -85,B 0,C 180,E1 -23438.42,E2 -23438.42} C_VEL
LIN {X 0,Y 211.897,Z 356.989,A -85,B 0,C 180,E1 -23438.358,E2 -23438.358} C_VEL
LIN {X 0,Y 210.147,Z 362.553,A -85,B 0,C 180,E1 -23438.607,E2 -23438.607} C_VEL
LIN {X 0,Y 205.99,Z 377.282,A -85,B 0,C 180,E1 -23439.856,E2 -23439.856} C_VEL
LIN {X 0,Y 201.574,Z 390.502,A -85,B 0,C 180,E1 -23441.392,E2 -23441.392} C_VEL
LIN {X 0,Y 196.572,Z 403.103,A -85,B 0,C 180,E1 -23443.242,E2 -23443.242} C_VEL
LIN {X 0,Y 190.711,Z 415.706,A -85,B 0,C 180,E1 -23445.558,E2 -23445.558} C_VEL
LIN {X 0,Y 184.767,Z 427.158,A -85,B 0,C 180,E1 -23448.268,E2 -23448.268} C_VEL
LIN {X 0,Y 179.309,Z 436.795,A -85,B 0,C 180,E1 -23451.162,E2 -23451.162} C_VEL
LIN {X 0,Y 173.645,Z 446.263,A -85,B 0,C 180,E1 -23454.778,E2 -23454.778} C_VEL
LIN {X 0,Y 168.477,Z 454.148,A -85,B 0,C 180,E1 -23458.571,E2 -23458.571} C_VEL
LIN {X 0,Y 163.633,Z 461.51,A -85,B 0,C 180,E1 -23463.194,E2 -23463.194} C_VEL
LIN {X 0,Y 159.915,Z 467.351,A -85,B 0,C 180,E1 -23468.064,E2 -23468.064} C_VEL
LIN {X 0,Y 157.793,Z 470.825,A -85,B 0,C 180,E1 -23471.834,E2 -23471.834} C_VEL
LIN {X 0,Y 155.809,Z 474.332,A -85,B 0,C 180,E1 -23476.966,E2 -23476.966} C_VEL
LIN {X 0,Y 154.846,Z 476.639,A -85,B 0,C 180,E1 -23482.174,E2 -23482.174} C_VEL
LIN {X 0,Y 154.627,Z 477.798,A -85,B 0,C 180,E1 -23487.395,E2 -23487.395} C_VEL
LIN {X 0,Y 154.623,Z 477.917,A -85,B 0,C 180,E1 -23490.593,E2 -23490.593} C_VEL
LIN {X 0,Y 154.679,Z 477.342,A -85,B 0,C 180,E1 -23495.214,E2 -23495.214} C_VEL
LIN {X 0,Y 155.218,Z 475.591,A -85,B 0,C 180,E1 -23500.434,E2 -23500.434} C_VEL
LIN {X 0,Y 156.603,Z 472.673,A -85,B 0,C 180,E1 -23505.621,E2 -23505.621} C_VEL
LIN {X 0,Y 159.106,Z 468.521,A -85,B 0,C 180,E1 -23510.694,E2 -23510.694} C_VEL
LIN {X 0,Y 162.553,Z 463.022,A -85,B 0,C 180,E1 -23515.617,E2 -23515.617} C_VEL
LIN {X 0,Y 167.201,Z 456.03,A -85,B 0,C 180,E1 -23520.291,E2 -23520.291} C_VEL
LIN {X 0,Y 172.123,Z 448.552,A -85,B 0,C 180,E1 -23524.155,E2 -23524.155} C_VEL
LIN {X 0,Y 177.495,Z 439.535,A -85,B 0,C 180,E1 -23527.858,E2 -23527.858} C_VEL
LIN {X 0,Y 183.85,Z 428.691,A -85,B 0,C 180,E1 -23531.255,E2 -23531.255} C_VEL
LIN {X 0,Y 190.16,Z 416.494,A -85,B 0,C 180,E1 -23534.234,E2 -23534.234} C_VEL
LIN {X 0,Y 196.041,Z 404.056,A -85,B 0,C 180,E1 -23536.548,E2 -23536.548} C_VEL
LIN {X 0,Y 201.405,Z 390.49,A -85,B 0,C 180,E1 -23538.562,E2 -23538.562} C_VEL
LIN {X 0,Y 205.999,Z 376.741,A -85,B 0,C 180,E1 -23540.141,E2 -23540.141} C_VEL
LIN {X 0,Y 209.854,Z 362.952,A -85,B 0,C 180,E1 -23541.328,E2 -23541.328} C_VEL
LIN {X 0,Y 213.211,Z 347.479,A -85,B 0,C 180,E1 -23542.289,E2 -23542.289} C_VEL
LIN {X 0,Y 215.483,Z 332.035,A -85,B 0,C 180,E1 -23542.951,E2 -23542.951} C_VEL
LIN {X 0,Y 220.864,Z 263.744,A -85,B 0,C 180,E1 -23544.824,E2 -23544.824} C_VEL
LIN {X 0,Y 216.093,Z 252.29,A -85,B 0,C 180,E1 -23547.338,E2 -23547.338} C_VEL
LIN {X 0,Y 211.054,Z 241.587,A -85,B 0,C 180,E1 -23550.24,E2 -23550.24} C_VEL
LIN {X 0,Y 206.53,Z 234.023,A -85,B 0,C 180,E1 -23553.067,E2 -23553.067} C_VEL
LIN {X 0,Y 201.25,Z 226.195,A -85,B 0,C 180,E1 -23556.867,E2 -23556.867} C_VEL
LIN {X 0,Y 198.003,Z 221.699,A -85,B 0,C 180,E1 -23559.617,E2 -23559.617} C_VEL
LIN {X 0,Y 194.824,Z 217.262,A -85,B 0,C 180,E1 -23562.822,E2 -23562.822} C_VEL
LIN {X 0,Y 192.42,Z 214.296,A -85,B 0,C 180,E1 -23565.727,E2 -23565.727} C_VEL
LIN {X 0,Y 191.587,Z 212.552,A -85,B 0,C 180,E1 -23567.016,E2 -23567.016} C_VEL
LIN {X 0,Y 189.177,Z 210.305,A -85,B 0,C 180,E1 -23571.185,E2 -23571.185} C_VEL
LIN {X 0,Y 188.078,Z 207.619,A -85,B 0,C 180,E1 -23574.64,E2 -23574.64} C_VEL
LIN {X 0,Y 187.329,Z 206.801,A -85,B 0,C 180,E1 -23580,E2 -23580} C_VEL
LIN {X 0,Y 188.103,Z 207.652,A -85,B 0,C 180,E1 -23585.629,E2 -23585.629} C_VEL
LIN {X 0,Y 189.99,Z 211.382,A -85,B 0,C 180,E1 -23590.659,E2 -23590.659} C_VEL
LIN {X 0,Y 191.632,Z 212.754,A -85,B 0,C 180,E1 -23593.251,E2 -23593.251} C_VEL
LIN {X 0,Y 193.735,Z 216.275,A -85,B 0,C 180,E1 -23596.158,E2 -23596.158} C_VEL
LIN {X 0,Y 195.301,Z 217.933,A -85,B 0,C 180,E1 -23597.879,E2 -23597.879} C_VEL
LIN {X 0,Y 197.964,Z 221.752,A -85,B 0,C 180,E1 -23600.535,E2 -23600.535} C_VEL
LIN {X 0,Y 199.239,Z 223.568,A -85,B 0,C 180,E1 -23601.671,E2 -23601.671} C_VEL
LIN {X 0,Y 202.133,Z 227.65,A -85,B 0,C 180,E1 -23604.011,E2 -23604.011} C_VEL
LIN {X 0,Y 205.373,Z 232.47,A -85,B 0,C 180,E1 -23606.349,E2 -23606.349} C_VEL
LIN {X 0,Y 210.175,Z 240.077,A -85,B 0,C 180,E1 -23609.414,E2 -23609.414} C_VEL
LIN {X 0,Y 215.313,Z 248.96,A -85,B 0,C 180,E1 -23612.311,E2 -23612.311} C_VEL
LIN {X 0,Y 218.521,Z 255.712,A -85,B 0,C 180,E1 -23614.013,E2 -23614.013} C_VEL
LIN {X 0,Y 221.003,Z 261.741,A -85,B 0,C 180,E1 -23615.293,E2 -23615.293} C_VEL
LIN {X 0,Y 215.574,Z 330.475,A -85,B 0,C 180,E1 -23617.194,E2 -23617.194} C_VEL
LIN {X 0,Y 213.33,Z 345.484,A -85,B 0,C 180,E1 -23617.849,E2 -23617.849} C_VEL
LIN {X 0,Y 210.177,Z 360.211,A -85,B 0,C 180,E1 -23618.782,E2 -23618.782} C_VEL
LIN {X 0,Y 206.401,Z 374.033,A -85,B 0,C 180,E1 -23619.992,E2 -23619.992} C_VEL
LIN {X 0,Y 202.294,Z 386.661,A -85,B 0,C 180,E1 -23621.452,E2 -23621.452} C_VEL
LIN {X 0,Y 197.052,Z 400.084,A -85,B 0,C 180,E1 -23623.39,E2 -23623.39} C_VEL
LIN {X 0,Y 191.236,Z 412.743,A -85,B 0,C 180,E1 -23625.713,E2 -23625.713} C_VEL
LIN {X 0,Y 185.34,Z 424.225,A -85,B 0,C 180,E1 -23628.426,E2 -23628.426} C_VEL
LIN {X 0,Y 179.303,Z 434.839,A -85,B 0,C 180,E1 -23631.622,E2 -23631.622} C_VEL
LIN {X 0,Y 174.282,Z 443.361,A -85,B 0,C 180,E1 -23634.926,E2 -23634.926} C_VEL
LIN {X 0,Y 169.113,Z 451.25,A -85,B 0,C 180,E1 -23638.703,E2 -23638.703} C_VEL
LIN {X 0,Y 164.19,Z 458.615,A -85,B 0,C 180,E1 -23643.292,E2 -23643.292} C_VEL
LIN {X 0,Y 160.37,Z 464.457,A -85,B 0,C 180,E1 -23648.13,E2 -23648.13} C_VEL
LIN {X 0,Y 158.19,Z 467.916,A -85,B 0,C 180,E1 -23651.881,E2 -23651.881} C_VEL
LIN {X 0,Y 156.128,Z 471.416,A -85,B 0,C 180,E1 -23656.993,E2 -23656.993} C_VEL
LIN {X 0,Y 154.986,Z 473.727,A -85,B 0,C 180,E1 -23662.181,E2 -23662.181} C_VEL
LIN {X 0,Y 154.667,Z 474.901,A -85,B 0,C 180,E1 -23667.396,E2 -23667.396} C_VEL
LIN {X 0,Y 154.657,Z 474.992,A -85,B 0,C 180,E1 -23671.301,E2 -23671.301} C_VEL
LIN {X 0,Y 154.757,Z 474.488,A -85,B 0,C 180,E1 -23675.211,E2 -23675.211} C_VEL
LIN {X 0,Y 155.433,Z 472.796,A -85,B 0,C 180,E1 -23680.42,E2 -23680.42} C_VEL
LIN {X 0,Y 156.955,Z 469.94,A -85,B 0,C 180,E1 -23685.585,E2 -23685.585} C_VEL
LIN {X 0,Y 159.585,Z 465.851,A -85,B 0,C 180,E1 -23690.629,E2 -23690.629} C_VEL
LIN {X 0,Y 163.122,Z 460.433,A -85,B 0,C 180,E1 -23695.521,E2 -23695.521} C_VEL
LIN {X 0,Y 167.73,Z 453.529,A -85,B 0,C 180,E1 -23700.186,E2 -23700.186} C_VEL
LIN {X 0,Y 172.615,Z 446.111,A -85,B 0,C 180,E1 -23704.044,E2 -23704.044} C_VEL
LIN {X 0,Y 177.293,Z 438.488,A -85,B 0,C 180,E1 -23707.211,E2 -23707.211} C_VEL
LIN {X 0,Y 183.385,Z 428.051,A -85,B 0,C 180,E1 -23710.655,E2 -23710.655} C_VEL
LIN {X 0,Y 189.113,Z 417.295,A -85,B 0,C 180,E1 -23713.434,E2 -23713.434} C_VEL
LIN {X 0,Y 194.771,Z 405.553,A -85,B 0,C 180,E1 -23715.821,E2 -23715.821} C_VEL
LIN {X 0,Y 200.204,Z 392.684,A -85,B 0,C 180,E1 -23717.878,E2 -23717.878} C_VEL
LIN {X 0,Y 205.173,Z 378.57,A -85,B 0,C 180,E1 -23719.654,E2 -23719.654} C_VEL
LIN {X 0,Y 209.15,Z 364.767,A -85,B 0,C 180,E1 -23720.993,E2 -23720.993} C_VEL
LIN {X 0,Y 212.753,Z 349.311,A -85,B 0,C 180,E1 -23722.062,E2 -23722.062} C_VEL
LIN {X 0,Y 215.294,Z 333.872,A -85,B 0,C 180,E1 -23722.813,E2 -23722.813} C_VEL
LIN {X 0,Y 217.16,Z 314.414,A -85,B 0,C 180,E1 -23723.41,E2 -23723.41} C_VEL
LIN {X 0,Y 221.178,Z 261.873,A -85,B 0,C 180,E1 -23724.835,E2 -23724.835} C_VEL
LIN {X 0,Y 216.576,Z 251.11,A -85,B 0,C 180,E1 -23727.247,E2 -23727.247} C_VEL
LIN {X 0,Y 210.697,Z 240.702,A -85,B 0,C 180,E1 -23730.528,E2 -23730.528} C_VEL
LIN {X 0,Y 205.457,Z 232.418,A -85,B 0,C 180,E1 -23733.87,E2 -23733.87} C_VEL
LIN {X 0,Y 201.166,Z 226.088,A -85,B 0,C 180,E1 -23737.051,E2 -23737.051} C_VEL
LIN {X 0,Y 198.056,Z 221.756,A -85,B 0,C 180,E1 -23739.724,E2 -23739.724} C_VEL
LIN {X 0,Y 195.348,Z 217.867,A -85,B 0,C 180,E1 -23742.463,E2 -23742.463} C_VEL
LIN {X 0,Y 192.35,Z 214.116,A -85,B 0,C 180,E1 -23746.126,E2 -23746.126} C_VEL
LIN {X 0,Y 191.624,Z 212.611,A -85,B 0,C 180,E1 -23747.287,E2 -23747.287} C_VEL
LIN {X 0,Y 189.154,Z 210.099,A -85,B 0,C 180,E1 -23751.856,E2 -23751.856} C_VEL
LIN {X 0,Y 188.207,Z 207.762,A -85,B 0,C 180,E1 -23755.18,E2 -23755.18} C_VEL
LIN {X 0,Y 187.659,Z 206.9,A -85,B 0,C 180,E1 -23760,E2 -23760} C_VEL
LIN {X 0,Y 188.197,Z 207.738,A -85,B 0,C 180,E1 -23764.685,E2 -23764.685} C_VEL
LIN {X 0,Y 190.593,Z 211.889,A -85,B 0,C 180,E1 -23771.028,E2 -23771.028} C_VEL
LIN {X 0,Y 191.799,Z 212.889,A -85,B 0,C 180,E1 -23772.902,E2 -23772.902} C_VEL
LIN {X 0,Y 194.116,Z 216.554,A -85,B 0,C 180,E1 -23776.087,E2 -23776.087} C_VEL
LIN {X 0,Y 195.446,Z 218.004,A -85,B 0,C 180,E1 -23777.558,E2 -23777.558} C_VEL
LIN {X 0,Y 198.245,Z 221.944,A -85,B 0,C 180,E1 -23780.356,E2 -23780.356} C_VEL
LIN {X 0,Y 202.279,Z 227.688,A -85,B 0,C 180,E1 -23783.736,E2 -23783.736} C_VEL
LIN {X 0,Y 205.727,Z 232.835,A -85,B 0,C 180,E1 -23786.229,E2 -23786.229} C_VEL
LIN {X 0,Y 210.165,Z 239.903,A -85,B 0,C 180,E1 -23789.073,E2 -23789.073} C_VEL
LIN {X 0,Y 213.871,Z 247.196,A -85,B 0,C 180,E1 -23791.273,E2 -23791.273} C_VEL
LIN {X 0,Y 219.117,Z 259.085,A -85,B 0,C 180,E1 -23794.145,E2 -23794.145} C_VEL
LIN {X 0,Y 221.043,Z 263.834,A -85,B 0,C 180,E1 -23795.137,E2 -23795.137} C_VEL
LIN {X 0,Y 215.573,Z 332.823,A -85,B 0,C 180,E1 -23797.035,E2 -23797.035} C_VEL
LIN {X 0,Y 213.264,Z 348.35,A -85,B 0,C 180,E1 -23797.729,E2 -23797.729} C_VEL
LIN {X 0,Y 210.147,Z 362.553,A -85,B 0,C 180,E1 -23798.607,E2 -23798.607} C_VEL
LIN {X 0,Y 208.292,Z 368.108,A -85,B 0,C 180,E1 -23798.901,E2 -23798.901} C_VEL
LIN {X 0,Y 203.917,Z 376.931,A -85,B 0,C 180,E1 -23799.086,E2 -23799.086} C_VEL
LIN {X 0,Y 199.21,Z 385.565,A -85,B 0,C 180,E1 -23799.384,E2 -23799.384} C_VEL
LIN {X 0,Y 196.844,Z 390.693,A -85,B 0,C 180,E1 -23799.869,E2 -23799.869} C_VEL
LIN {X 0,Y 191.204,Z 404.33,A -85,B 0,C 180,E1 -23801.899,E2 -23801.899} C_VEL
LIN {X 0,Y 185.159,Z 416.713,A -85,B 0,C 180,E1 -23804.239,E2 -23804.239} C_VEL
LIN {X 0,Y 178.537,Z 428.85,A -85,B 0,C 180,E1 -23807.232,E2 -23807.232} C_VEL
LIN {X 0,Y 172.795,Z 438.367,A -85,B 0,C 180,E1 -23810.24,E2 -23810.24} C_VEL
LIN {X 0,Y 167.049,Z 447.432,A -85,B 0,C 180,E1 -23813.914,E2 -23813.914} C_VEL
LIN {X 0,Y 161.058,Z 456.103,A -85,B 0,C 180,E1 -23818.423,E2 -23818.423} C_VEL
LIN {X 0,Y 156.17,Z 463.06,A -85,B 0,C 180,E1 -23823.255,E2 -23823.255} C_VEL
LIN {X 0,Y 152.451,Z 468.531,A -85,B 0,C 180,E1 -23828.358,E2 -23828.358} C_VEL
LIN {X 0,Y 149.739,Z 472.666,A -85,B 0,C 180,E1 -23833.644,E2 -23833.644} C_VEL
LIN {X 0,Y 148.217,Z 475.566,A -85,B 0,C 180,E1 -23839.066,E2 -23839.066} C_VEL
LIN {X 0,Y 147.606,Z 477.294,A -85,B 0,C 180,E1 -23844.536,E2 -23844.536} C_VEL
LIN {X 0,Y 147.587,Z 477.884,A -85,B 0,C 180,E1 -23850,E2 -23850} C_VEL
LIN {X 0,Y 147.606,Z 477.276,A -85,B 0,C 180,E1 -23855.464,E2 -23855.464} C_VEL
LIN {X 0,Y 148.215,Z 475.524,A -85,B 0,C 180,E1 -23860.933,E2 -23860.933} C_VEL
LIN {X 0,Y 149.727,Z 472.605,A -85,B 0,C 180,E1 -23866.358,E2 -23866.358} C_VEL
LIN {X 0,Y 152.437,Z 468.453,A -85,B 0,C 180,E1 -23871.644,E2 -23871.644} C_VEL
LIN {X 0,Y 156.128,Z 462.954,A -85,B 0,C 180,E1 -23876.753,E2 -23876.753} C_VEL
LIN {X 0,Y 161.053,Z 455.961,A -85,B 0,C 180,E1 -23881.578,E2 -23881.578} C_VEL
LIN {X 0,Y 166.256,Z 448.484,A -85,B 0,C 180,E1 -23885.538,E2 -23885.538} C_VEL
LIN {X 0,Y 171.015,Z 440.818,A -85,B 0,C 180,E1 -23888.808,E2 -23888.808} C_VEL
LIN {X 0,Y 177.555,Z 430.257,A -85,B 0,C 180,E1 -23892.291,E2 -23892.291} C_VEL
LIN {X 0,Y 183.552,Z 419.409,A -85,B 0,C 180,E1 -23895.1,E2 -23895.1} C_VEL
LIN {X 0,Y 189.521,Z 407.566,A -85,B 0,C 180,E1 -23897.478,E2 -23897.478} C_VEL
LIN {X 0,Y 195.077,Z 394.751,A -85,B 0,C 180,E1 -23899.518,E2 -23899.518} C_VEL
LIN {X 0,Y 199.728,Z 382.045,A -85,B 0,C 180,E1 -23901.127,E2 -23901.127} C_VEL
LIN {X 0,Y 203.927,Z 368.531,A -85,B 0,C 180,E1 -23902.434,E2 -23902.434} C_VEL
LIN {X 0,Y 207.687,Z 353.554,A -85,B 0,C 180,E1 -23903.483,E2 -23903.483} C_VEL
LIN {X 0,Y 210.388,Z 338.731,A -85,B 0,C 180,E1 -23904.225,E2 -23904.225} C_VEL
LIN {X 0,Y 212.126,Z 322.885,A -85,B 0,C 180,E1 -23904.765,E2 -23904.765} C_VEL
LIN {X 0,Y 216.637,Z 266.466,A -85,B 0,C 180,E1 -23906.279,E2 -23906.279} C_VEL
LIN {X 0,Y 212.678,Z 256.817,A -85,B 0,C 180,E1 -23908.511,E2 -23908.511} C_VEL
LIN {X 0,Y 208.284,Z 247.089,A -85,B 0,C 180,E1 -23911.209,E2 -23911.209} C_VEL
LIN {X 0,Y 204.119,Z 239.928,A -85,B 0,C 180,E1 -23913.96,E2 -23913.96} C_VEL
LIN {X 0,Y 199.335,Z 232.561,A -85,B 0,C 180,E1 -23917.591,E2 -23917.591} C_VEL
LIN {X 0,Y 196.241,Z 228.134,A -85,B 0,C 180,E1 -23920.348,E2 -23920.348} C_VEL
LIN {X 0,Y 193.395,Z 223.961,A -85,B 0,C 180,E1 -23923.371,E2 -23923.371} C_VEL
LIN {X 0,Y 191.023,Z 220.883,A -85,B 0,C 180,E1 -23926.402,E2 -23926.402} C_VEL
LIN {X 0,Y 190.193,Z 219.344,A -85,B 0,C 180,E1 -23927.733,E2 -23927.733} C_VEL
LIN {X 0,Y 187.885,Z 216.717,A -85,B 0,C 180,E1 -23932.207,E2 -23932.207} C_VEL
LIN {X 0,Y 187.073,Z 214.53,A -85,B 0,C 180,E1 -23935.151,E2 -23935.151} C_VEL
LIN {X 0,Y 186.466,Z 213.823,A -85,B 0,C 180,E1 -23940,E2 -23940} C_VEL
LIN {X 0,Y 187.031,Z 214.481,A -85,B 0,C 180,E1 -23944.85,E2 -23944.85} C_VEL
LIN {X 0,Y 189.275,Z 218.667,A -85,B 0,C 180,E1 -23950.97,E2 -23950.97} C_VEL
LIN {X 0,Y 190.462,Z 219.765,A -85,B 0,C 180,E1 -23952.878,E2 -23952.878} C_VEL
LIN {X 0,Y 192.582,Z 223.243,A -85,B 0,C 180,E1 -23955.885,E2 -23955.885} C_VEL
LIN {X 0,Y 193.848,Z 224.7,A -85,B 0,C 180,E1 -23957.336,E2 -23957.336} C_VEL
LIN {X 0,Y 196.461,Z 228.472,A -85,B 0,C 180,E1 -23960.042,E2 -23960.042} C_VEL
LIN {X 0,Y 200.153,Z 233.939,A -85,B 0,C 180,E1 -23963.268,E2 -23963.268} C_VEL
LIN {X 0,Y 204.239,Z 240.207,A -85,B 0,C 180,E1 -23966.307,E2 -23966.307} C_VEL
LIN {X 0,Y 209.367,Z 248.965,A -85,B 0,C 180,E1 -23969.629,E2 -23969.629} C_VEL
LIN {X 0,Y 213.683,Z 257.071,A -85,B 0,C 180,E1 -23972.118,E2 -23972.118} C_VEL
LIN {X 0,Y 216.713,Z 264.323,A -85,B 0,C 180,E1 -23973.803,E2 -23973.803} C_VEL
LIN {X 0,Y 211.377,Z 330.487,A -85,B 0,C 180,E1 -23975.661,E2 -23975.661} C_VEL
LIN {X 0,Y 209.057,Z 345.56,A -85,B 0,C 180,E1 -23976.315,E2 -23976.315} C_VEL
LIN {X 0,Y 205.817,Z 360.285,A -85,B 0,C 180,E1 -23977.246,E2 -23977.246} C_VEL
LIN {X 0,Y 201.915,Z 374.105,A -85,B 0,C 180,E1 -23978.45,E2 -23978.45} C_VEL
LIN {X 0,Y 197.384,Z 387.501,A -85,B 0,C 180,E1 -23980.005,E2 -23980.005} C_VEL
LIN {X 0,Y 192.223,Z 400.155,A -85,B 0,C 180,E1 -23981.846,E2 -23981.846} C_VEL
LIN {X 0,Y 186.211,Z 412.813,A -85,B 0,C 180,E1 -23984.184,E2 -23984.184} C_VEL
LIN {X 0,Y 180.085,Z 424.294,A -85,B 0,C 180,E1 -23986.925,E2 -23986.925} C_VEL
LIN {X 0,Y 174.35,Z 433.958,A -85,B 0,C 180,E1 -23989.838,E2 -23989.838} C_VEL
LIN {X 0,Y 168.499,Z 443.43,A -85,B 0,C 180,E1 -23993.533,E2 -23993.533} C_VEL
LIN {X 0,Y 163.052,Z 451.319,A -85,B 0,C 180,E1 -23997.399,E2 -23997.399} C_VEL
LIN {X 0,Y 157.84,Z 458.683,A -85,B 0,C 180,E1 -24002.126,E2 -24002.126} C_VEL
LIN {X 0,Y 153.752,Z 464.525,A -85,B 0,C 180,E1 -24007.137,E2 -24007.137} C_VEL
LIN {X 0,Y 151.434,Z 467.983,A -85,B 0,C 180,E1 -24011.043,E2 -24011.043} C_VEL
LIN {X 0,Y 149.169,Z 471.484,A -85,B 0,C 180,E1 -24016.375,E2 -24016.375} C_VEL
LIN {X 0,Y 147.952,Z 473.794,A -85,B 0,C 180,E1 -24021.807,E2 -24021.807} C_VEL
LIN {X 0,Y 147.571,Z 474.968,A -85,B 0,C 180,E1 -24027.27,E2 -24027.27} C_VEL
LIN {X 0,Y 147.597,Z 475.101,A -85,B 0,C 180,E1 -24030.613,E2 -24030.613} C_VEL
LIN {X 0,Y 147.689,Z 474.554,A -85,B 0,C 180,E1 -24035.461,E2 -24035.461} C_VEL
LIN {X 0,Y 148.416,Z 472.862,A -85,B 0,C 180,E1 -24040.919,E2 -24040.919} C_VEL
LIN {X 0,Y 150.083,Z 470.006,A -85,B 0,C 180,E1 -24046.318,E2 -24046.318} C_VEL
LIN {X 0,Y 152.892,Z 465.917,A -85,B 0,C 180,E1 -24051.576,E2 -24051.576} C_VEL
LIN {X 0,Y 156.703,Z 460.498,A -85,B 0,C 180,E1 -24056.647,E2 -24056.647} C_VEL
LIN {X 0,Y 161.591,Z 453.594,A -85,B 0,C 180,E1 -24061.461,E2 -24061.461} C_VEL
LIN {X 0,Y 166.769,Z 446.175,A -85,B 0,C 180,E1 -24065.412,E2 -24065.412} C_VEL
LIN {X 0,Y 172.206,Z 437.654,A -85,B 0,C 180,E1 -24069.006,E2 -24069.006} C_VEL
LIN {X 0,Y 178.035,Z 428.115,A -85,B 0,C 180,E1 -24072.151,E2 -24072.151} C_VEL
LIN {X 0,Y 184.002,Z 417.359,A -85,B 0,C 180,E1 -24074.96,E2 -24074.96} C_VEL
LIN {X 0,Y 189.884,Z 405.615,A -85,B 0,C 180,E1 -24077.359,E2 -24077.359} C_VEL
LIN {X 0,Y 195.366,Z 393.106,A -85,B 0,C 180,E1 -24079.371,E2 -24079.371} C_VEL
LIN {X 0,Y 200.068,Z 380.395,A -85,B 0,C 180,E1 -24081.006,E2 -24081.006} C_VEL
LIN {X 0,Y 204.153,Z 367.084,A -85,B 0,C 180,E1 -24082.353,E2 -24082.353} C_VEL
LIN {X 0,Y 207.839,Z 352.413,A -85,B 0,C 180,E1 -24083.427,E2 -24083.427} C_VEL
LIN {X 0,Y 210.721,Z 336.704,A -85,B 0,C 180,E1 -24084.234,E2 -24084.234} C_VEL
LIN {X 0,Y 212.428,Z 321.621,A -85,B 0,C 180,E1 -24084.752,E2 -24084.752} C_VEL
LIN {X 0,Y 216.931,Z 264.619,A -85,B 0,C 180,E1 -24086.303,E2 -24086.303} C_VEL
LIN {X 0,Y 213.013,Z 255.408,A -85,B 0,C 180,E1 -24088.498,E2 -24088.498} C_VEL
LIN {X 0,Y 207.698,Z 245.816,A -85,B 0,C 180,E1 -24091.661,E2 -24091.661} C_VEL
LIN {X 0,Y 203.095,Z 238.304,A -85,B 0,C 180,E1 -24094.782,E2 -24094.782} C_VEL
LIN {X 0,Y 199.055,Z 232.193,A -85,B 0,C 180,E1 -24097.951,E2 -24097.951} C_VEL
LIN {X 0,Y 196.367,Z 228.294,A -85,B 0,C 180,E1 -24100.395,E2 -24100.395} C_VEL
LIN {X 0,Y 193.453,Z 224.071,A -85,B 0,C 180,E1 -24103.524,E2 -24103.524} C_VEL
LIN {X 0,Y 190.955,Z 220.659,A -85,B 0,C 180,E1 -24106.836,E2 -24106.836} C_VEL
LIN {X 0,Y 190.249,Z 219.383,A -85,B 0,C 180,E1 -24108.007,E2 -24108.007} C_VEL
LIN {X 0,Y 187.945,Z 216.667,A -85,B 0,C 180,E1 -24112.749,E2 -24112.749} C_VEL
LIN {X 0,Y 187.226,Z 214.647,A -85,B 0,C 180,E1 -24115.694,E2 -24115.694} C_VEL
LIN {X 0,Y 186.793,Z 213.95,A -85,B 0,C 180,E1 -24120,E2 -24120} C_VEL
LIN {X 0,Y 187.241,Z 214.691,A -85,B 0,C 180,E1 -24124.305,E2 -24124.305} C_VEL
LIN {X 0,Y 189.735,Z 219.008,A -85,B 0,C 180,E1 -24131.078,E2 -24131.078} C_VEL
LIN {X 0,Y 190.627,Z 219.838,A -85,B 0,C 180,E1 -24132.509,E2 -24132.509} C_VEL
LIN {X 0,Y 192.848,Z 223.403,A -85,B 0,C 180,E1 -24135.68,E2 -24135.68} C_VEL
LIN {X 0,Y 194.08,Z 224.917,A -85,B 0,C 180,E1 -24137.111,E2 -24137.111} C_VEL
LIN {X 0,Y 197.491,Z 229.842,A -85,B 0,C 180,E1 -24140.574,E2 -24140.574} C_VEL
LIN {X 0,Y 200.291,Z 233.996,A -85,B 0,C 180,E1 -24142.984,E2 -24142.984} C_VEL
LIN {X 0,Y 204.502,Z 240.431,A -85,B 0,C 180,E1 -24146.124,E2 -24146.124} C_VEL
LIN {X 0,Y 208.736,Z 247.817,A -85,B 0,C 180,E1 -24148.917,E2 -24148.917} C_VEL
LIN {X 0,Y 213.101,Z 257.462,A -85,B 0,C 180,E1 -24151.584,E2 -24151.584} C_VEL
LIN {X 0,Y 216.812,Z 266.625,A -85,B 0,C 180,E1 -24153.681,E2 -24153.681} C_VEL
LIN {X 0,Y 211.389,Z 332.662,A -85,B 0,C 180,E1 -24155.495,E2 -24155.495} C_VEL
LIN {X 0,Y 209.002,Z 348.293,A -85,B 0,C 180,E1 -24156.192,E2 -24156.192} C_VEL
LIN {X 0,Y 205.694,Z 362.886,A -85,B 0,C 180,E1 -24157.094,E2 -24157.094} C_VEL
LIN {X 0,Y 201.503,Z 377.222,A -85,B 0,C 180,E1 -24158.302,E2 -24158.302} C_VEL
LIN {X 0,Y 196.844,Z 390.693,A -85,B 0,C 180,E1 -24159.869,E2 -24159.869} C_VEL
LIN {X 0,Y 194.352,Z 395.822,A -85,B 0,C 180,E1 -24160.412,E2 -24160.412} C_VEL
LIN {X 0,Y 188.908,Z 403.968,A -85,B 0,C 180,E1 -24161.013,E2 -24161.013} C_VEL
LIN {X 0,Y 183.274,Z 411.702,A -85,B 0,C 180,E1 -24161.756,E2 -24161.756} C_VEL
LIN {X 0,Y 180.51,Z 416.188,A -85,B 0,C 180,E1 -24162.524,E2 -24162.524} C_VEL
LIN {X 0,Y 174.385,Z 427.03,A -85,B 0,C 180,E1 -24165.148,E2 -24165.148} C_VEL
LIN {X 0,Y 168.389,Z 436.666,A -85,B 0,C 180,E1 -24168.103,E2 -24168.103} C_VEL
LIN {X 0,Y 162.082,Z 446.195,A -85,B 0,C 180,E1 -24171.878,E2 -24171.878} C_VEL
LIN {X 0,Y 156.458,Z 454.017,A -85,B 0,C 180,E1 -24175.841,E2 -24175.841} C_VEL
LIN {X 0,Y 150.979,Z 461.379,A -85,B 0,C 180,E1 -24180.74,E2 -24180.74} C_VEL
LIN {X 0,Y 146.594,Z 467.361,A -85,B 0,C 180,E1 -24186.123,E2 -24186.123} C_VEL
LIN {X 0,Y 144.28,Z 470.693,A -85,B 0,C 180,E1 -24190.063,E2 -24190.063} C_VEL
LIN {X 0,Y 141.914,Z 474.2,A -85,B 0,C 180,E1 -24195.663,E2 -24195.663} C_VEL
LIN {X 0,Y 140.748,Z 476.507,A -85,B 0,C 180,E1 -24201.385,E2 -24201.385} C_VEL
LIN {X 0,Y 140.428,Z 477.665,A -85,B 0,C 180,E1 -24207.131,E2 -24207.131} C_VEL
LIN {X 0,Y 140.484,Z 477.817,A -85,B 0,C 180,E1 -24210,E2 -24210} C_VEL
LIN {X 0,Y 140.527,Z 477.209,A -85,B 0,C 180,E1 -24215.74,E2 -24215.74} C_VEL
LIN {X 0,Y 141.201,Z 475.457,A -85,B 0,C 180,E1 -24221.484,E2 -24221.484} C_VEL
LIN {X 0,Y 142.884,Z 472.538,A -85,B 0,C 180,E1 -24227.165,E2 -24227.165} C_VEL
LIN {X 0,Y 145.812,Z 468.385,A -85,B 0,C 180,E1 -24232.68,E2 -24232.68} C_VEL
LIN {X 0,Y 149.767,Z 462.886,A -85,B 0,C 180,E1 -24237.986,E2 -24237.986} C_VEL
LIN {X 0,Y 154.976,Z 455.893,A -85,B 0,C 180,E1 -24242.969,E2 -24242.969} C_VEL
LIN {X 0,Y 160.488,Z 448.415,A -85,B 0,C 180,E1 -24247.023,E2 -24247.023} C_VEL
LIN {X 0,Y 165.508,Z 440.75,A -85,B 0,C 180,E1 -24250.358,E2 -24250.358} C_VEL
LIN {X 0,Y 172.35,Z 430.188,A -85,B 0,C 180,E1 -24253.885,E2 -24253.885} C_VEL
LIN {X 0,Y 178.588,Z 419.339,A -85,B 0,C 180,E1 -24256.722,E2 -24256.722} C_VEL
LIN {X 0,Y 184.786,Z 407.496,A -85,B 0,C 180,E1 -24259.105,E2 -24259.105} C_VEL
LIN {X 0,Y 190.701,Z 394.26,A -85,B 0,C 180,E1 -24261.207,E2 -24261.207} C_VEL
LIN {X 0,Y 195.954,Z 380.206,A -85,B 0,C 180,E1 -24262.94,E2 -24262.94} C_VEL
LIN {X 0,Y 200.325,Z 366.201,A -85,B 0,C 180,E1 -24264.222,E2 -24264.222} C_VEL
LIN {X 0,Y 204.001,Z 351.19,A -85,B 0,C 180,E1 -24265.229,E2 -24265.229} C_VEL
LIN {X 0,Y 206.734,Z 335.702,A -85,B 0,C 180,E1 -24265.935,E2 -24265.935} C_VEL
LIN {X 0,Y 208.798,Z 315.232,A -85,B 0,C 180,E1 -24266.539,E2 -24266.539} C_VEL
LIN {X 0,Y 212.523,Z 269.247,A -85,B 0,C 180,E1 -24267.8,E2 -24267.8} C_VEL
LIN {X 0,Y 209.032,Z 260.584,A -85,B 0,C 180,E1 -24269.923,E2 -24269.923} C_VEL
LIN {X 0,Y 205.304,Z 252.005,A -85,B 0,C 180,E1 -24272.39,E2 -24272.39} C_VEL
LIN {X 0,Y 201.045,Z 244.693,A -85,B 0,C 180,E1 -24275.405,E2 -24275.405} C_VEL
LIN {X 0,Y 196.824,Z 238.086,A -85,B 0,C 180,E1 -24278.874,E2 -24278.874} C_VEL
LIN {X 0,Y 194.573,Z 234.662,A -85,B 0,C 180,E1 -24281.03,E2 -24281.03} C_VEL
LIN {X 0,Y 191.868,Z 230.614,A -85,B 0,C 180,E1 -24284.055,E2 -24284.055} C_VEL
LIN {X 0,Y 189.458,Z 227.06,A -85,B 0,C 180,E1 -24287.412,E2 -24287.412} C_VEL
LIN {X 0,Y 189,Z 226.208,A -85,B 0,C 180,E1 -24288.199,E2 -24288.199} C_VEL
LIN {X 0,Y 186.795,Z 223.48,A -85,B 0,C 180,E1 -24292.788,E2 -24292.788} C_VEL
LIN {X 0,Y 186.081,Z 221.466,A -85,B 0,C 180,E1 -24295.668,E2 -24295.668} C_VEL
LIN {X 0,Y 185.601,Z 220.874,A -85,B 0,C 180,E1 -24300,E2 -24300} C_VEL
LIN {X 0,Y 186.166,Z 221.549,A -85,B 0,C 180,E1 -24304.873,E2 -24304.873} C_VEL
LIN {X 0,Y 187.95,Z 225.34,A -85,B 0,C 180,E1 -24310.163,E2 -24310.163} C_VEL
LIN {X 0,Y 189.225,Z 226.601,A -85,B 0,C 180,E1 -24312.365,E2 -24312.365} C_VEL
LIN {X 0,Y 191.305,Z 230.055,A -85,B 0,C 180,E1 -24315.447,E2 -24315.447} C_VEL
LIN {X 0,Y 192.465,Z 231.557,A -85,B 0,C 180,E1 -24316.849,E2 -24316.849} C_VEL
LIN {X 0,Y 195.695,Z 236.409,A -85,B 0,C 180,E1 -24320.259,E2 -24320.259} C_VEL
LIN {X 0,Y 198.667,Z 241.02,A -85,B 0,C 180,E1 -24322.901,E2 -24322.901} C_VEL
LIN {X 0,Y 202.099,Z 246.449,A -85,B 0,C 180,E1 -24325.556,E2 -24325.556} C_VEL
LIN {X 0,Y 207.149,Z 255.368,A -85,B 0,C 180,E1 -24328.981,E2 -24328.981} C_VEL
LIN {X 0,Y 210.866,Z 262.808,A -85,B 0,C 180,E1 -24331.244,E2 -24331.244} C_VEL
LIN {X 0,Y 212.614,Z 267.23,A -85,B 0,C 180,E1 -24332.29,E2 -24332.29} C_VEL
LIN {X 0,Y 207.314,Z 330.637,A -85,B 0,C 180,E1 -24334.072,E2 -24334.072} C_VEL
LIN {X 0,Y 204.933,Z 345.637,A -85,B 0,C 180,E1 -24334.716,E2 -24334.716} C_VEL
LIN {X 0,Y 201.601,Z 360.36,A -85,B 0,C 180,E1 -24335.64,E2 -24335.64} C_VEL
LIN {X 0,Y 197.571,Z 374.178,A -85,B 0,C 180,E1 -24336.835,E2 -24336.835} C_VEL
LIN {X 0,Y 192.633,Z 388.28,A -85,B 0,C 180,E1 -24338.478,E2 -24338.478} C_VEL
LIN {X 0,Y 186.986,Z 401.515,A -85,B 0,C 180,E1 -24340.438,E2 -24340.438} C_VEL
LIN {X 0,Y 180.776,Z 413.95,A -85,B 0,C 180,E1 -24342.794,E2 -24342.794} C_VEL
LIN {X 0,Y 174.96,Z 424.363,A -85,B 0,C 180,E1 -24345.335,E2 -24345.335} C_VEL
LIN {X 0,Y 168.965,Z 434.027,A -85,B 0,C 180,E1 -24348.278,E2 -24348.278} C_VEL
LIN {X 0,Y 163.629,Z 442.272,A -85,B 0,C 180,E1 -24351.48,E2 -24351.48} C_VEL
LIN {X 0,Y 157.831,Z 450.382,A -85,B 0,C 180,E1 -24355.407,E2 -24355.407} C_VEL
LIN {X 0,Y 152.862,Z 457.076,A -85,B 0,C 180,E1 -24359.62,E2 -24359.62} C_VEL
LIN {X 0,Y 148.15,Z 463.271,A -85,B 0,C 180,E1 -24364.726,E2 -24364.726} C_VEL
LIN {X 0,Y 144.684,Z 468.051,A -85,B 0,C 180,E1 -24370.122,E2 -24370.122} C_VEL
LIN {X 0,Y 142.237,Z 471.551,A -85,B 0,C 180,E1 -24375.697,E2 -24375.697} C_VEL
LIN {X 0,Y 140.915,Z 473.861,A -85,B 0,C 180,E1 -24381.395,E2 -24381.395} C_VEL
LIN {X 0,Y 140.49,Z 475.034,A -85,B 0,C 180,E1 -24387.133,E2 -24387.133} C_VEL
LIN {X 0,Y 140.524,Z 475.19,A -85,B 0,C 180,E1 -24390,E2 -24390} C_VEL
LIN {X 0,Y 140.62,Z 474.621,A -85,B 0,C 180,E1 -24395.737,E2 -24395.737} C_VEL
LIN {X 0,Y 141.42,Z 472.928,A -85,B 0,C 180,E1 -24401.466,E2 -24401.466} C_VEL
LIN {X 0,Y 143.24,Z 470.072,A -85,B 0,C 180,E1 -24407.121,E2 -24407.121} C_VEL
LIN {X 0,Y 146.252,Z 465.983,A -85,B 0,C 180,E1 -24412.609,E2 -24412.609} C_VEL
LIN {X 0,Y 150.353,Z 460.564,A -85,B 0,C 180,E1 -24417.868,E2 -24417.868} C_VEL
LIN {X 0,Y 155.523,Z 453.659,A -85,B 0,C 180,E1 -24422.839,E2 -24422.839} C_VEL
LIN {X 0,Y 161.02,Z 446.24,A -85,B 0,C 180,E1 -24426.88,E2 -24426.88} C_VEL
LIN {X 0,Y 167.393,Z 436.767,A -85,B 0,C 180,E1 -24430.91,E2 -24430.91} C_VEL
LIN {X 0,Y 173.839,Z 426.554,A -85,B 0,C 180,E1 -24434.218,E2 -24434.218} C_VEL
LIN {X 0,Y 180.679,Z 414.477,A -85,B 0,C 180,E1 -24437.24,E2 -24437.24} C_VEL
LIN {X 0,Y 186.859,Z 402.145,A -85,B 0,C 180,E1 -24439.608,E2 -24439.608} C_VEL
LIN {X 0,Y 192.675,Z 388.602,A -85,B 0,C 180,E1 -24441.631,E2 -24441.631} C_VEL
LIN {X 0,Y 197.457,Z 375.153,A -85,B 0,C 180,E1 -24443.21,E2 -24443.21} C_VEL
LIN {X 0,Y 201.501,Z 361.498,A -85,B 0,C 180,E1 -24444.4,E2 -24444.4} C_VEL
LIN {X 0,Y 204.99,Z 346.377,A -85,B 0,C 180,E1 -24445.369,E2 -24445.369} C_VEL
LIN {X 0,Y 207.479,Z 330.847,A -85,B 0,C 180,E1 -24446.055,E2 -24446.055} C_VEL
LIN {X 0,Y 212.805,Z 268.696,A -85,B 0,C 180,E1 -24447.756,E2 -24447.756} C_VEL
LIN {X 0,Y 212.823,Z 267.436,A -85,B 0,C 180,E1 -24447.826,E2 -24447.826} C_VEL
LIN {X 0,Y 209.852,Z 260.386,A -85,B 0,C 180,E1 -24449.607,E2 -24449.607} C_VEL
LIN {X 0,Y 205.204,Z 251.671,A -85,B 0,C 180,E1 -24452.544,E2 -24452.544} C_VEL
LIN {X 0,Y 200.695,Z 244.002,A -85,B 0,C 180,E1 -24455.789,E2 -24455.789} C_VEL
LIN {X 0,Y 197.204,Z 238.555,A -85,B 0,C 180,E1 -24458.688,E2 -24458.688} C_VEL
LIN {X 0,Y 194.646,Z 234.729,A -85,B 0,C 180,E1 -24461.139,E2 -24461.139} C_VEL
LIN {X 0,Y 191.955,Z 230.69,A -85,B 0,C 180,E1 -24464.196,E2 -24464.196} C_VEL
LIN {X 0,Y 189.591,Z 227.187,A -85,B 0,C 180,E1 -24467.557,E2 -24467.557} C_VEL
LIN {X 0,Y 189.065,Z 226.265,A -85,B 0,C 180,E1 -24468.474,E2 -24468.474} C_VEL
LIN {X 0,Y 186.822,Z 223.308,A -85,B 0,C 180,E1 -24473.52,E2 -24473.52} C_VEL
LIN {X 0,Y 186.255,Z 221.571,A -85,B 0,C 180,E1 -24476.214,E2 -24476.214} C_VEL
LIN {X 0,Y 185.957,Z 221.052,A -85,B 0,C 180,E1 -24481.083,E2 -24481.083} C_VEL
LIN {X 0,Y 186.445,Z 222.051,A -85,B 0,C 180,E1 -24484.73,E2 -24484.73} C_VEL
LIN {X 0,Y 188.362,Z 225.665,A -85,B 0,C 180,E1 -24490.208,E2 -24490.208} C_VEL
LIN {X 0,Y 189.424,Z 226.739,A -85,B 0,C 180,E1 -24492.046,E2 -24492.046} C_VEL
LIN {X 0,Y 191.691,Z 230.345,A -85,B 0,C 180,E1 -24495.388,E2 -24495.388} C_VEL
LIN {X 0,Y 192.662,Z 231.701,A -85,B 0,C 180,E1 -24496.576,E2 -24496.576} C_VEL
LIN {X 0,Y 195.883,Z 236.512,A -85,B 0,C 180,E1 -24499.997,E2 -24499.997} C_VEL
LIN {X 0,Y 198.38,Z 240.332,A -85,B 0,C 180,E1 -24502.248,E2 -24502.248} C_VEL
LIN {X 0,Y 202.262,Z 246.529,A -85,B 0,C 180,E1 -24505.302,E2 -24505.302} C_VEL
LIN {X 0,Y 206.093,Z 253.43,A -85,B 0,C 180,E1 -24507.97,E2 -24507.97} C_VEL
LIN {X 0,Y 210.286,Z 263.189,A -85,B 0,C 180,E1 -24510.692,E2 -24510.692} C_VEL
LIN {X 0,Y 212.723,Z 269.405,A -85,B 0,C 180,E1 -24512.167,E2 -24512.167} C_VEL
LIN {X 0,Y 207.329,Z 332.724,A -85,B 0,C 180,E1 -24513.901,E2 -24513.901} C_VEL
LIN {X 0,Y 204.887,Z 348.236,A -85,B 0,C 180,E1 -24514.589,E2 -24514.589} C_VEL
LIN {X 0,Y 201.33,Z 363.451,A -85,B 0,C 180,E1 -24515.532,E2 -24515.532} C_VEL
LIN {X 0,Y 197.185,Z 377.161,A -85,B 0,C 180,E1 -24516.684,E2 -24516.684} C_VEL
LIN {X 0,Y 192.132,Z 391.215,A -85,B 0,C 180,E1 -24518.314,E2 -24518.314} C_VEL
LIN {X 0,Y 186.487,Z 404.374,A -85,B 0,C 180,E1 -24520.292,E2 -24520.292} C_VEL
LIN {X 0,Y 180.51,Z 416.188,A -85,B 0,C 180,E1 -24522.524,E2 -24522.524} C_VEL
LIN {X 0,Y 177.665,Z 420.67,A -85,B 0,C 180,E1 -24523.358,E2 -24523.358} C_VEL
LIN {X 0,Y 171.517,Z 427.702,A -85,B 0,C 180,E1 -24524.467,E2 -24524.467} C_VEL
LIN {X 0,Y 165.198,Z 434.296,A -85,B 0,C 180,E1 -24525.781,E2 -24525.781} C_VEL
LIN {X 0,Y 162.144,Z 438.091,A -85,B 0,C 180,E1 -24526.948,E2 -24526.948} C_VEL
LIN {X 0,Y 155.674,Z 447.301,A -85,B 0,C 180,E1 -24530.799,E2 -24530.799} C_VEL
LIN {X 0,Y 149.796,Z 454.962,A -85,B 0,C 180,E1 -24534.919,E2 -24534.919} C_VEL
LIN {X 0,Y 144.765,Z 461.313,A -85,B 0,C 180,E1 -24539.353,E2 -24539.353} C_VEL
LIN {X 0,Y 140.727,Z 466.472,A -85,B 0,C 180,E1 -24544.017,E2 -24544.017} C_VEL
LIN {X 0,Y 137.561,Z 470.627,A -85,B 0,C 180,E1 -24549.045,E2 -24549.045} C_VEL
LIN {X 0,Y 134.985,Z 474.133,A -85,B 0,C 180,E1 -24554.91,E2 -24554.91} C_VEL
LIN {X 0,Y 133.702,Z 476.44,A -85,B 0,C 180,E1 -24560.927,E2 -24560.927} C_VEL
LIN {X 0,Y 133.33,Z 477.599,A -85,B 0,C 180,E1 -24566.978,E2 -24566.978} C_VEL
LIN {X 0,Y 133.39,Z 477.751,A -85,B 0,C 180,E1 -24570,E2 -24570} C_VEL
LIN {X 0,Y 133.443,Z 477.142,A -85,B 0,C 180,E1 -24576.046,E2 -24576.046} C_VEL
LIN {X 0,Y 134.213,Z 475.389,A -85,B 0,C 180,E1 -24582.09,E2 -24582.09} C_VEL
LIN {X 0,Y 136.078,Z 472.47,A -85,B 0,C 180,E1 -24588.052,E2 -24588.052} C_VEL
LIN {X 0,Y 139.239,Z 468.317,A -85,B 0,C 180,E1 -24593.815,E2 -24593.815} C_VEL
LIN {X 0,Y 143.485,Z 462.817,A -85,B 0,C 180,E1 -24599.328,E2 -24599.328} C_VEL
LIN {X 0,Y 149.005,Z 455.824,A -85,B 0,C 180,E1 -24604.471,E2 -24604.471} C_VEL
LIN {X 0,Y 154.828,Z 448.346,A -85,B 0,C 180,E1 -24608.619,E2 -24608.619} C_VEL
LIN {X 0,Y 160.135,Z 440.681,A -85,B 0,C 180,E1 -24612.013,E2 -24612.013} C_VEL
LIN {X 0,Y 167.285,Z 430.119,A -85,B 0,C 180,E1 -24615.578,E2 -24615.578} C_VEL
LIN {X 0,Y 173.772,Z 419.269,A -85,B 0,C 180,E1 -24618.435,E2 -24618.435} C_VEL
LIN {X 0,Y 180.207,Z 407.426,A -85,B 0,C 180,E1 -24620.815,E2 -24620.815} C_VEL
LIN {X 0,Y 185.953,Z 395.058,A -85,B 0,C 180,E1 -24622.792,E2 -24622.792} C_VEL
LIN {X 0,Y 191.115,Z 381.901,A -85,B 0,C 180,E1 -24624.451,E2 -24624.451} C_VEL
LIN {X 0,Y 195.595,Z 368.384,A -85,B 0,C 180,E1 -24625.733,E2 -24625.733} C_VEL
LIN {X 0,Y 199.546,Z 353.402,A -85,B 0,C 180,E1 -24626.77,E2 -24626.77} C_VEL
LIN {X 0,Y 202.485,Z 338.182,A -85,B 0,C 180,E1 -24627.496,E2 -24627.496} C_VEL
LIN {X 0,Y 204.317,Z 322.039,A -85,B 0,C 180,E1 -24628.04,E2 -24628.04} C_VEL
LIN {X 0,Y 208.555,Z 272.025,A -85,B 0,C 180,E1 -24629.384,E2 -24629.384} C_VEL
LIN {X 0,Y 204.572,Z 261.942,A -85,B 0,C 180,E1 -24632.047,E2 -24632.047} C_VEL
LIN {X 0,Y 202.103,Z 256.447,A -85,B 0,C 180,E1 -24633.82,E2 -24633.82} C_VEL
LIN {X 0,Y 197.823,Z 248.896,A -85,B 0,C 180,E1 -24637.134,E2 -24637.134} C_VEL
LIN {X 0,Y 193.332,Z 241.663,A -85,B 0,C 180,E1 -24641.316,E2 -24641.316} C_VEL
LIN {X 0,Y 190.374,Z 237.216,A -85,B 0,C 180,E1 -24644.75,E2 -24644.75} C_VEL
LIN {X 0,Y 188.114,Z 233.583,A -85,B 0,C 180,E1 -24648.143,E2 -24648.143} C_VEL
LIN {X 0,Y 186.878,Z 232.202,A -85,B 0,C 180,E1 -24650.394,E2 -24650.394} C_VEL
LIN {X 0,Y 185.216,Z 228.533,A -85,B 0,C 180,E1 -24655.648,E2 -24655.648} C_VEL
LIN {X 0,Y 184.738,Z 227.899,A -85,B 0,C 180,E1 -24660,E2 -24660} C_VEL
LIN {X 0,Y 185.241,Z 228.529,A -85,B 0,C 180,E1 -24664.625,E2 -24664.625} C_VEL
LIN {X 0,Y 186.728,Z 232.067,A -85,B 0,C 180,E1 -24669.478,E2 -24669.478} C_VEL
LIN {X 0,Y 188.049,Z 233.528,A -85,B 0,C 180,E1 -24671.93,E2 -24671.93} C_VEL
LIN {X 0,Y 190.136,Z 237.011,A -85,B 0,C 180,E1 -24675.133,E2 -24675.133} C_VEL
LIN {X 0,Y 191.122,Z 238.443,A -85,B 0,C 180,E1 -24676.385,E2 -24676.385} C_VEL
LIN {X 0,Y 194.008,Z 242.936,A -85,B 0,C 180,E1 -24679.578,E2 -24679.578} C_VEL
LIN {X 0,Y 196.988,Z 247.664,A -85,B 0,C 180,E1 -24682.345,E2 -24682.345} C_VEL
LIN {X 0,Y 201.114,Z 254.723,A -85,B 0,C 180,E1 -24685.64,E2 -24685.64} C_VEL
LIN {X 0,Y 205.861,Z 263.658,A -85,B 0,C 180,E1 -24688.918,E2 -24688.918} C_VEL
LIN {X 0,Y 208.559,Z 269.739,A -85,B 0,C 180,E1 -24690.643,E2 -24690.643} C_VEL
LIN {X 0,Y 208.699,Z 270.178,A -85,B 0,C 180,E1 -24690.736,E2 -24690.736} C_VEL
LIN {X 0,Y 203.506,Z 330.096,A -85,B 0,C 180,E1 -24692.393,E2 -24692.393} C_VEL
LIN {X 0,Y 200.979,Z 345.714,A -85,B 0,C 180,E1 -24693.054,E2 -24693.054} C_VEL
LIN {X 0,Y 197.549,Z 360.434,A -85,B 0,C 180,E1 -24693.966,E2 -24693.966} C_VEL
LIN {X 0,Y 193.402,Z 374.251,A -85,B 0,C 180,E1 -24695.152,E2 -24695.152} C_VEL
LIN {X 0,Y 188.651,Z 387.375,A -85,B 0,C 180,E1 -24696.655,E2 -24696.655} C_VEL
LIN {X 0,Y 183.05,Z 400.296,A -85,B 0,C 180,E1 -24698.531,E2 -24698.531} C_VEL
LIN {X 0,Y 176.597,Z 412.953,A -85,B 0,C 180,E1 -24700.875,E2 -24700.875} C_VEL
LIN {X 0,Y 169.977,Z 424.433,A -85,B 0,C 180,E1 -24703.65,E2 -24703.65} C_VEL
LIN {X 0,Y 163.713,Z 434.096,A -85,B 0,C 180,E1 -24706.618,E2 -24706.618} C_VEL
LIN {X 0,Y 158.1,Z 442.341,A -85,B 0,C 180,E1 -24709.867,E2 -24709.867} C_VEL
LIN {X 0,Y 151.979,Z 450.451,A -85,B 0,C 180,E1 -24713.871,E2 -24713.871} C_VEL
LIN {X 0,Y 146.733,Z 457.144,A -85,B 0,C 180,E1 -24718.206,E2 -24718.206} C_VEL
LIN {X 0,Y 141.697,Z 463.339,A -85,B 0,C 180,E1 -24723.488,E2 -24723.488} C_VEL
LIN {X 0,Y 137.982,Z 468.119,A -85,B 0,C 180,E1 -24729.112,E2 -24729.112} C_VEL
LIN {X 0,Y 135.336,Z 471.618,A -85,B 0,C 180,E1 -24734.951,E2 -24734.951} C_VEL
LIN {X 0,Y 133.879,Z 473.928,A -85,B 0,C 180,E1 -24740.939,E2 -24740.939} C_VEL
LIN {X 0,Y 133.402,Z 475.101,A -85,B 0,C 180,E1 -24746.98,E2 -24746.98} C_VEL
LIN {X 0,Y 133.449,Z 475.256,A -85,B 0,C 180,E1 -24750,E2 -24750} C_VEL
LIN {X 0,Y 133.548,Z 474.687,A -85,B 0,C 180,E1 -24756.042,E2 -24756.042} C_VEL
LIN {X 0,Y 134.449,Z 472.994,A -85,B 0,C 180,E1 -24762.069,E2 -24762.069} C_VEL
LIN {X 0,Y 136.426,Z 470.138,A -85,B 0,C 180,E1 -24768.005,E2 -24768.005} C_VEL
LIN {X 0,Y 139.671,Z 466.049,A -85,B 0,C 180,E1 -24773.738,E2 -24773.738} C_VEL
LIN {X 0,Y 144.058,Z 460.629,A -85,B 0,C 180,E1 -24779.2,E2 -24779.2} C_VEL
LIN {X 0,Y 149.563,Z 453.725,A -85,B 0,C 180,E1 -24784.325,E2 -24784.325} C_VEL
LIN {X 0,Y 155.381,Z 446.305,A -85,B 0,C 180,E1 -24788.457,E2 -24788.457} C_VEL
LIN {X 0,Y 161.627,Z 437.426,A -85,B 0,C 180,E1 -24792.336,E2 -24792.336} C_VEL
LIN {X 0,Y 167.734,Z 428.243,A -85,B 0,C 180,E1 -24795.422,E2 -24795.422} C_VEL
LIN {X 0,Y 174.212,Z 417.485,A -85,B 0,C 180,E1 -24798.273,E2 -24798.273} C_VEL
LIN {X 0,Y 180.552,Z 405.741,A -85,B 0,C 180,E1 -24800.682,E2 -24800.682} C_VEL
LIN {X 0,Y 186.584,Z 392.84,A -85,B 0,C 180,E1 -24802.745,E2 -24802.745} C_VEL
LIN {X 0,Y 192.043,Z 378.753,A -85,B 0,C 180,E1 -24804.515,E2 -24804.515} C_VEL
LIN {X 0,Y 196.463,Z 364.944,A -85,B 0,C 180,E1 -24805.817,E2 -24805.817} C_VEL
LIN {X 0,Y 200.368,Z 349.48,A -85,B 0,C 180,E1 -24806.87,E2 -24806.87} C_VEL
LIN {X 0,Y 203.064,Z 334.664,A -85,B 0,C 180,E1 -24807.569,E2 -24807.569} C_VEL
LIN {X 0,Y 205.127,Z 315.209,A -85,B 0,C 180,E1 -24808.17,E2 -24808.17} C_VEL
LIN {X 0,Y 208.938,Z 270.461,A -85,B 0,C 180,E1 -24809.364,E2 -24809.364} C_VEL
LIN {X 0,Y 206.597,Z 264.952,A -85,B 0,C 180,E1 -24810.864,E2 -24810.864} C_VEL
LIN {X 0,Y 202.3,Z 256.675,A -85,B 0,C 180,E1 -24813.777,E2 -24813.777} C_VEL
LIN {X 0,Y 198.11,Z 249.236,A -85,B 0,C 180,E1 -24817.031,E2 -24817.031} C_VEL
LIN {X 0,Y 194.708,Z 243.927,A -85,B 0,C 180,E1 -24820.083,E2 -24820.083} C_VEL
LIN {X 0,Y 193.137,Z 241.399,A -85,B 0,C 180,E1 -24821.708,E2 -24821.708} C_VEL
LIN {X 0,Y 190.585,Z 237.397,A -85,B 0,C 180,E1 -24824.753,E2 -24824.753} C_VEL
LIN {X 0,Y 188.395,Z 234.063,A -85,B 0,C 180,E1 -24828.023,E2 -24828.023} C_VEL
LIN {X 0,Y 187.893,Z 233.157,A -85,B 0,C 180,E1 -24828.948,E2 -24828.948} C_VEL
LIN {X 0,Y 185.834,Z 230.232,A -85,B 0,C 180,E1 -24833.894,E2 -24833.894} C_VEL
LIN {X 0,Y 185.387,Z 228.653,A -85,B 0,C 180,E1 -24836.196,E2 -24836.196} C_VEL
LIN {X 0,Y 185.062,Z 228.05,A -85,B 0,C 180,E1 -24840,E2 -24840} C_VEL
LIN {X 0,Y 185.45,Z 228.789,A -85,B 0,C 180,E1 -24844.074,E2 -24844.074} C_VEL
LIN {X 0,Y 187.228,Z 232.517,A -85,B 0,C 180,E1 -24849.725,E2 -24849.725} C_VEL
LIN {X 0,Y 188.238,Z 233.602,A -85,B 0,C 180,E1 -24851.576,E2 -24851.576} C_VEL
LIN {X 0,Y 190.443,Z 237.176,A -85,B 0,C 180,E1 -24854.97,E2 -24854.97} C_VEL
LIN {X 0,Y 193.937,Z 242.529,A -85,B 0,C 180,E1 -24859.035,E2 -24859.035} C_VEL
LIN {X 0,Y 196.928,Z 247.4,A -85,B 0,C 180,E1 -24861.881,E2 -24861.881} C_VEL
LIN {X 0,Y 200.212,Z 252.856,A -85,B 0,C 180,E1 -24864.573,E2 -24864.573} C_VEL
LIN {X 0,Y 203.452,Z 259.01,A -85,B 0,C 180,E1 -24866.967,E2 -24866.967} C_VEL
LIN {X 0,Y 207.242,Z 268.216,A -85,B 0,C 180,E1 -24869.593,E2 -24869.593} C_VEL
LIN {X 0,Y 208.794,Z 272.288,A -85,B 0,C 180,E1 -24870.604,E2 -24870.604} C_VEL
LIN {X 0,Y 203.553,Z 332.017,A -85,B 0,C 180,E1 -24872.223,E2 -24872.223} C_VEL
LIN {X 0,Y 201.075,Z 347.575,A -85,B 0,C 180,E1 -24872.893,E2 -24872.893} C_VEL
LIN {X 0,Y 197.614,Z 362.206,A -85,B 0,C 180,E1 -24873.766,E2 -24873.766} C_VEL
LIN {X 0,Y 193.032,Z 377.101,A -85,B 0,C 180,E1 -24874.996,E2 -24874.996} C_VEL
LIN {X 0,Y 188.04,Z 390.537,A -85,B 0,C 180,E1 -24876.53,E2 -24876.53} C_VEL
LIN {X 0,Y 182.436,Z 403.337,A -85,B 0,C 180,E1 -24878.433,E2 -24878.433} C_VEL
LIN {X 0,Y 176.096,Z 415.517,A -85,B 0,C 180,E1 -24880.686,E2 -24880.686} C_VEL
LIN {X 0,Y 169.409,Z 426.966,A -85,B 0,C 180,E1 -24883.448,E2 -24883.448} C_VEL
LIN {X 0,Y 163.139,Z 436.601,A -85,B 0,C 180,E1 -24886.427,E2 -24886.427} C_VEL
LIN {X 0,Y 162.144,Z 438.091,A -85,B 0,C 180,E1 -24886.948,E2 -24886.948} C_VEL
LIN {X 0,Y 159.108,Z 441.772,A -85,B 0,C 180,E1 -24888.21,E2 -24888.21} C_VEL
LIN {X 0,Y 152.727,Z 447.514,A -85,B 0,C 180,E1 -24890.063,E2 -24890.063} C_VEL
LIN {X 0,Y 146.322,Z 452.788,A -85,B 0,C 180,E1 -24892.155,E2 -24892.155} C_VEL
LIN {X 0,Y 143.323,Z 455.711,A -85,B 0,C 180,E1 -24893.786,E2 -24893.786} C_VEL
LIN {X 0,Y 137.297,Z 462.863,A -85,B 0,C 180,E1 -24899.21,E2 -24899.21} C_VEL
LIN {X 0,Y 132.707,Z 468.333,A -85,B 0,C 180,E1 -24904.933,E2 -24904.933} C_VEL
LIN {X 0,Y 129.326,Z 472.468,A -85,B 0,C 180,E1 -24910.97,E2 -24910.97} C_VEL
LIN {X 0,Y 127.253,Z 475.367,A -85,B 0,C 180,E1 -24917.237,E2 -24917.237} C_VEL
LIN {X 0,Y 126.366,Z 477.095,A -85,B 0,C 180,E1 -24923.613,E2 -24923.613} C_VEL
LIN {X 0,Y 126.307,Z 477.685,A -85,B 0,C 180,E1 -24930,E2 -24930} C_VEL
LIN {X 0,Y 126.366,Z 477.076,A -85,B 0,C 180,E1 -24936.386,E2 -24936.386} C_VEL
LIN {X 0,Y 127.25,Z 475.322,A -85,B 0,C 180,E1 -24942.763,E2 -24942.763} C_VEL
LIN {X 0,Y 129.31,Z 472.403,A -85,B 0,C 180,E1 -24949.032,E2 -24949.032} C_VEL
LIN {X 0,Y 132.7,Z 468.249,A -85,B 0,C 180,E1 -24955.068,E2 -24955.068} C_VEL
LIN {X 0,Y 137.279,Z 462.749,A -85,B 0,C 180,E1 -24960.794,E2 -24960.794} C_VEL
LIN {X 0,Y 143.158,Z 455.755,A -85,B 0,C 180,E1 -24966.094,E2 -24966.094} C_VEL
LIN {X 0,Y 149.284,Z 448.277,A -85,B 0,C 180,E1 -24970.34,E2 -24970.34} C_VEL
LIN {X 0,Y 153.884,Z 441.967,A -85,B 0,C 180,E1 -24973.241,E2 -24973.241} C_VEL
LIN {X 0,Y 161.264,Z 431.68,A -85,B 0,C 180,E1 -24976.885,E2 -24976.885} C_VEL
LIN {X 0,Y 167.968,Z 421.153,A -85,B 0,C 180,E1 -24979.783,E2 -24979.783} C_VEL
LIN {X 0,Y 174.563,Z 409.704,A -85,B 0,C 180,E1 -24982.196,E2 -24982.196} C_VEL
LIN {X 0,Y 180.466,Z 397.87,A -85,B 0,C 180,E1 -24984.174,E2 -24984.174} C_VEL
LIN {X 0,Y 186.431,Z 383.596,A -85,B 0,C 180,E1 -24986.032,E2 -24986.032} C_VEL
LIN {X 0,Y 191.346,Z 369.439,A -85,B 0,C 180,E1 -24987.403,E2 -24987.403} C_VEL
LIN {X 0,Y 195.58,Z 354.089,A -85,B 0,C 180,E1 -24988.464,E2 -24988.464} C_VEL
LIN {X 0,Y 198.631,Z 338.928,A -85,B 0,C 180,E1 -24989.195,E2 -24989.195} C_VEL
LIN {X 0,Y 200.581,Z 322.778,A -85,B 0,C 180,E1 -24989.736,E2 -24989.736} C_VEL
LIN {X 0,Y 204.706,Z 276.267,A -85,B 0,C 180,E1 -24990.949,E2 -24990.949} C_VEL
LIN {X 0,Y 204.673,Z 274.63,A -85,B 0,C 180,E1 -24991.082,E2 -24991.082} C_VEL
LIN {X 0,Y 200.335,Z 263.512,A -85,B 0,C 180,E1 -24994.288,E2 -24994.288} C_VEL
LIN {X 0,Y 196.539,Z 256.466,A -85,B 0,C 180,E1 -24997.324,E2 -24997.324} C_VEL
LIN {X 0,Y 193.156,Z 250.722,A -85,B 0,C 180,E1 -25000.463,E2 -25000.463} C_VEL
LIN {X 0,Y 191.154,Z 247.44,A -85,B 0,C 180,E1 -25002.619,E2 -25002.619} C_VEL
LIN {X 0,Y 189.01,Z 243.914,A -85,B 0,C 180,E1 -25005.327,E2 -25005.327} C_VEL
LIN {X 0,Y 186.649,Z 239.955,A -85,B 0,C 180,E1 -25009.149,E2 -25009.149} C_VEL
LIN {X 0,Y 184.597,Z 236.808,A -85,B 0,C 180,E1 -25014.265,E2 -25014.265} C_VEL
LIN {X 0,Y 184.237,Z 235.484,A -85,B 0,C 180,E1 -25016.173,E2 -25016.173} C_VEL
LIN {X 0,Y 183.872,Z 234.95,A -85,B 0,C 180,E1 -25020,E2 -25020} C_VEL
LIN {X 0,Y 184.304,Z 235.628,A -85,B 0,C 180,E1 -25024.374,E2 -25024.374} C_VEL
LIN {X 0,Y 185.861,Z 239.224,A -85,B 0,C 180,E1 -25029.523,E2 -25029.523} C_VEL
LIN {X 0,Y 186.833,Z 240.34,A -85,B 0,C 180,E1 -25031.39,E2 -25031.39} C_VEL
LIN {X 0,Y 189.173,Z 244.171,A -85,B 0,C 180,E1 -25035.074,E2 -25035.074} C_VEL
LIN {X 0,Y 192.44,Z 249.609,A -85,B 0,C 180,E1 -25038.982,E2 -25038.982} C_VEL
LIN {X 0,Y 195.852,Z 255.203,A -85,B 0,C 180,E1 -25042.248,E2 -25042.248} C_VEL
LIN {X 0,Y 200.397,Z 263.651,A -85,B 0,C 180,E1 -25045.936,E2 -25045.936} C_VEL
LIN {X 0,Y 204.593,Z 272.282,A -85,B 0,C 180,E1 -25048.887,E2 -25048.887} C_VEL
LIN {X 0,Y 204.902,Z 273.128,A -85,B 0,C 180,E1 -25049.104,E2 -25049.104} C_VEL
LIN {X 0,Y 199.727,Z 330.714,A -85,B 0,C 180,E1 -25050.696,E2 -25050.696} C_VEL
LIN {X 0,Y 197.203,Z 345.791,A -85,B 0,C 180,E1 -25051.328,E2 -25051.328} C_VEL
LIN {X 0,Y 193.677,Z 360.508,A -85,B 0,C 180,E1 -25052.227,E2 -25052.227} C_VEL
LIN {X 0,Y 189.395,Z 374.324,A -85,B 0,C 180,E1 -25053.392,E2 -25053.392} C_VEL
LIN {X 0,Y 184.255,Z 388.035,A -85,B 0,C 180,E1 -25054.954,E2 -25054.954} C_VEL
LIN {X 0,Y 178.092,Z 401.656,A -85,B 0,C 180,E1 -25056.954,E2 -25056.954} C_VEL
LIN {X 0,Y 171.437,Z 414.09,A -85,B 0,C 180,E1 -25059.306,E2 -25059.306} C_VEL
LIN {X 0,Y 165.131,Z 424.502,A -85,B 0,C 180,E1 -25061.858,E2 -25061.858} C_VEL
LIN {X 0,Y 158.59,Z 434.165,A -85,B 0,C 180,E1 -25064.842,E2 -25064.842} C_VEL
LIN {X 0,Y 152.704,Z 442.409,A -85,B 0,C 180,E1 -25068.138,E2 -25068.138} C_VEL
LIN {X 0,Y 146.267,Z 450.519,A -85,B 0,C 180,E1 -25072.22,E2 -25072.22} C_VEL
LIN {X 0,Y 140.716,Z 457.212,A -85,B 0,C 180,E1 -25076.675,E2 -25076.675} C_VEL
LIN {X 0,Y 135.308,Z 463.407,A -85,B 0,C 180,E1 -25082.13,E2 -25082.13} C_VEL
LIN {X 0,Y 131.331,Z 468.186,A -85,B 0,C 180,E1 -25088.001,E2 -25088.001} C_VEL
LIN {X 0,Y 128.467,Z 471.685,A -85,B 0,C 180,E1 -25094.125,E2 -25094.125} C_VEL
LIN {X 0,Y 126.866,Z 473.994,A -85,B 0,C 180,E1 -25100.434,E2 -25100.434} C_VEL
LIN {X 0,Y 126.309,Z 475.167,A -85,B 0,C 180,E1 -25106.81,E2 -25106.81} C_VEL
LIN {X 0,Y 126.36,Z 475.323,A -85,B 0,C 180,E1 -25110,E2 -25110} C_VEL
LIN {X 0,Y 126.47,Z 474.753,A -85,B 0,C 180,E1 -25116.381,E2 -25116.381} C_VEL
LIN {X 0,Y 127.474,Z 473.06,A -85,B 0,C 180,E1 -25122.74,E2 -25122.74} C_VEL
LIN {X 0,Y 129.648,Z 470.204,A -85,B 0,C 180,E1 -25128.981,E2 -25128.981} C_VEL
LIN {X 0,Y 133.159,Z 466.115,A -85,B 0,C 180,E1 -25134.976,E2 -25134.976} C_VEL
LIN {X 0,Y 137.848,Z 460.695,A -85,B 0,C 180,E1 -25140.653,E2 -25140.653} C_VEL
LIN {X 0,Y 143.727,Z 453.79,A -85,B 0,C 180,E1 -25145.929,E2 -25145.929} C_VEL
LIN {X 0,Y 149.864,Z 446.369,A -85,B 0,C 180,E1 -25150.152,E2 -25150.152} C_VEL
LIN {X 0,Y 155.979,Z 438.072,A -85,B 0,C 180,E1 -25153.869,E2 -25153.869} C_VEL
LIN {X 0,Y 162.812,Z 428.306,A -85,B 0,C 180,E1 -25157.208,E2 -25157.208} C_VEL
LIN {X 0,Y 169.565,Z 417.549,A -85,B 0,C 180,E1 -25160.065,E2 -25160.065} C_VEL
LIN {X 0,Y 176.128,Z 405.803,A -85,B 0,C 180,E1 -25162.474,E2 -25162.474} C_VEL
LIN {X 0,Y 182.661,Z 392.227,A -85,B 0,C 180,E1 -25164.62,E2 -25164.62} C_VEL
LIN {X 0,Y 188.01,Z 378.813,A -85,B 0,C 180,E1 -25166.277,E2 -25166.277} C_VEL
LIN {X 0,Y 192.566,Z 365.003,A -85,B 0,C 180,E1 -25167.564,E2 -25167.564} C_VEL
LIN {X 0,Y 196.583,Z 349.536,A -85,B 0,C 180,E1 -25168.6,E2 -25168.6} C_VEL
LIN {X 0,Y 199.431,Z 334.088,A -85,B 0,C 180,E1 -25169.319,E2 -25169.319} C_VEL
LIN {X 0,Y 201.578,Z 314.229,A -85,B 0,C 180,E1 -25169.906,E2 -25169.906} C_VEL
LIN {X 0,Y 205.139,Z 273.354,A -85,B 0,C 180,E1 -25171.003,E2 -25171.003} C_VEL
LIN {X 0,Y 201.997,Z 266.564,A -85,B 0,C 180,E1 -25173.178,E2 -25173.178} C_VEL
LIN {X 0,Y 197.599,Z 258.087,A -85,B 0,C 180,E1 -25176.576,E2 -25176.576} C_VEL
LIN {X 0,Y 193.821,Z 251.616,A -85,B 0,C 180,E1 -25179.988,E2 -25179.988} C_VEL
LIN {X 0,Y 191.419,Z 247.757,A -85,B 0,C 180,E1 -25182.54,E2 -25182.54} C_VEL
LIN {X 0,Y 189.211,Z 244.124,A -85,B 0,C 180,E1 -25185.342,E2 -25185.342} C_VEL
LIN {X 0,Y 186.95,Z 240.287,A -85,B 0,C 180,E1 -25189.029,E2 -25189.029} C_VEL
LIN {X 0,Y 184.683,Z 236.566,A -85,B 0,C 180,E1 -25195.088,E2 -25195.088} C_VEL
LIN {X 0,Y 184.432,Z 235.57,A -85,B 0,C 180,E1 -25196.723,E2 -25196.723} C_VEL
LIN {X 0,Y 184.225,Z 235.16,A -85,B 0,C 180,E1 -25201.093,E2 -25201.093} C_VEL
LIN {X 0,Y 184.565,Z 236.015,A -85,B 0,C 180,E1 -25204.094,E2 -25204.094} C_VEL
LIN {X 0,Y 186.365,Z 239.649,A -85,B 0,C 180,E1 -25209.77,E2 -25209.77} C_VEL
LIN {X 0,Y 187.03,Z 240.408,A -85,B 0,C 180,E1 -25211.035,E2 -25211.035} C_VEL
LIN {X 0,Y 189.834,Z 245.094,A -85,B 0,C 180,E1 -25215.412,E2 -25215.412} C_VEL
LIN {X 0,Y 192.652,Z 249.715,A -85,B 0,C 180,E1 -25218.731,E2 -25218.731} C_VEL
LIN {X 0,Y 195.399,Z 254.283,A -85,B 0,C 180,E1 -25221.425,E2 -25221.425} C_VEL
LIN {X 0,Y 199.33,Z 261.309,A -85,B 0,C 180,E1 -25224.735,E2 -25224.735} C_VEL
LIN {X 0,Y 201.333,Z 265.67,A -85,B 0,C 180,E1 -25226.288,E2 -25226.288} C_VEL
LIN {X 0,Y 204.995,Z 275.135,A -85,B 0,C 180,E1 -25228.963,E2 -25228.963} C_VEL
LIN {X 0,Y 199.785,Z 332.456,A -85,B 0,C 180,E1 -25230.514,E2 -25230.514} C_VEL
LIN {X 0,Y 197.178,Z 348.122,A -85,B 0,C 180,E1 -25231.192,E2 -25231.192} C_VEL
LIN {X 0,Y 193.426,Z 363.332,A -85,B 0,C 180,E1 -25232.108,E2 -25232.108} C_VEL
LIN {X 0,Y 189.047,Z 377.04,A -85,B 0,C 180,E1 -25233.232,E2 -25233.232} C_VEL
LIN {X 0,Y 183.893,Z 390.469,A -85,B 0,C 180,E1 -25234.746,E2 -25234.746} C_VEL
LIN {X 0,Y 177.954,Z 403.58,A -85,B 0,C 180,E1 -25236.688,E2 -25236.688} C_VEL
LIN {X 0,Y 170.949,Z 416.523,A -85,B 0,C 180,E1 -25239.106,E2 -25239.106} C_VEL
LIN {X 0,Y 163.456,Z 428.657,A -85,B 0,C 180,E1 -25242.125,E2 -25242.125} C_VEL
LIN {X 0,Y 155.972,Z 439.452,A -85,B 0,C 180,E1 -25245.699,E2 -25245.699} C_VEL
LIN {X 0,Y 149.298,Z 448.446,A -85,B 0,C 180,E1 -25249.664,E2 -25249.664} C_VEL
LIN {X 0,Y 143.323,Z 455.711,A -85,B 0,C 180,E1 -25253.786,E2 -25253.786} C_VEL
LIN {X 0,Y 140.406,Z 458.544,A -85,B 0,C 180,E1 -25255.522,E2 -25255.522} C_VEL
LIN {X 0,Y 134.333,Z 462.765,A -85,B 0,C 180,E1 -25258.283,E2 -25258.283} C_VEL
LIN {X 0,Y 128.544,Z 466.418,A -85,B 0,C 180,E1 -25261.409,E2 -25261.409} C_VEL
LIN {X 0,Y 126.164,Z 468.36,A -85,B 0,C 180,E1 -25263.679,E2 -25263.679} C_VEL
LIN {X 0,Y 122.601,Z 472.402,A -85,B 0,C 180,E1 -25269.882,E2 -25269.882} C_VEL
LIN {X 0,Y 120.279,Z 475.3,A -85,B 0,C 180,E1 -25276.483,E2 -25276.483} C_VEL
LIN {X 0,Y 119.279,Z 477.028,A -85,B 0,C 180,E1 -25283.232,E2 -25283.232} C_VEL
LIN {X 0,Y 119.226,Z 477.618,A -85,B 0,C 180,E1 -25290,E2 -25290} C_VEL
LIN {X 0,Y 119.279,Z 477.009,A -85,B 0,C 180,E1 -25296.767,E2 -25296.767} C_VEL
LIN {X 0,Y 120.275,Z 475.255,A -85,B 0,C 180,E1 -25303.517,E2 -25303.517} C_VEL
LIN {X 0,Y 122.557,Z 472.335,A -85,B 0,C 180,E1 -25310.125,E2 -25310.125} C_VEL
LIN {X 0,Y 126.234,Z 468.181,A -85,B 0,C 180,E1 -25316.448,E2 -25316.448} C_VEL
LIN {X 0,Y 131.173,Z 462.681,A -85,B 0,C 180,E1 -25322.397,E2 -25322.397} C_VEL
LIN {X 0,Y 137.439,Z 455.687,A -85,B 0,C 180,E1 -25327.852,E2 -25327.852} C_VEL
LIN {X 0,Y 143.869,Z 448.208,A -85,B 0,C 180,E1 -25332.197,E2 -25332.197} C_VEL
LIN {X 0,Y 148.769,Z 441.899,A -85,B 0,C 180,E1 -25335.122,E2 -25335.122} C_VEL
LIN {X 0,Y 156.478,Z 431.611,A -85,B 0,C 180,E1 -25338.79,E2 -25338.79} C_VEL
LIN {X 0,Y 163.446,Z 421.083,A -85,B 0,C 180,E1 -25341.696,E2 -25341.696} C_VEL
LIN {X 0,Y 170.289,Z 409.634,A -85,B 0,C 180,E1 -25344.09,E2 -25344.09} C_VEL
LIN {X 0,Y 175.987,Z 398.611,A -85,B 0,C 180,E1 -25345.928,E2 -25345.928} C_VEL
LIN {X 0,Y 181.894,Z 385.174,A -85,B 0,C 180,E1 -25347.694,E2 -25347.694} C_VEL
